LIN {X 0,Y 354.882,Z 183.277,A -85,B 0,C 180,E1 -13338.473,E2 -13338.473} C_VEL
LIN {X 0,Y 354.834,Z 183.282,A -85,B 0,C 180,E1 -13342.106,E2 -13342.106} C_VEL
LIN {X 0,Y 354.874,Z 183.277,A -85,B 0,C 180,E1 -13345.829,E2 -13345.829} C_VEL
LIN {X 0,Y 354.83,Z 183.283,A -85,B 0,C 180,E1 -13349.681,E2 -13349.681} C_VEL
LIN {X 0,Y 354.784,Z 183.288,A -85,B 0,C 180,E1 -13353.704,E2 -13353.704} C_VEL
LIN {X 0,Y 354.778,Z 183.294,A -85,B 0,C 180,E1 -13356.462,E2 -13356.462} C_VEL
LIN {X 0,Y 354.805,Z 183.286,A -85,B 0,C 180,E1 -13359.426,E2 -13359.426} C_VEL
LIN {X 0,Y 354.823,Z 183.285,A -85,B 0,C 180,E1 -13362.879,E2 -13362.879} C_VEL
LIN {X 0,Y 354.859,Z 183.284,A -85,B 0,C 180,E1 -13366.123,E2 -13366.123} C_VEL
LIN {X 0,Y 354.921,Z 183.373,A -85,B 0,C 180,E1 -13367.406,E2 -13367.406} C_VEL
LIN {X 0,Y 355.833,Z 189.151,A -85,B 0,C 180,E1 -13371.532,E2 -13371.532} C_VEL
LIN {X 0,Y 356.15,Z 192.833,A -85,B 0,C 180,E1 -13374.004,E2 -13374.004} C_VEL
LIN {X 0,Y 355.889,Z 196.663,A -85,B 0,C 180,E1 -13376.435,E2 -13376.435} C_VEL
LIN {X 0,Y 355.418,Z 202.03,A -85,B 0,C 180,E1 -13379.723,E2 -13379.723} C_VEL
LIN {X 0,Y 354.813,Z 207.607,A -85,B 0,C 180,E1 -13383.043,E2 -13383.043} C_VEL
LIN {X 0,Y 354.335,Z 213.763,A -85,B 0,C 180,E1 -13386.631,E2 -13386.631} C_VEL
LIN {X 0,Y 353.966,Z 219.424,A -85,B 0,C 180,E1 -13389.822,E2 -13389.822} C_VEL
LIN {X 0,Y 356.521,Z 232.448,A -85,B 0,C 180,E1 -13390.431,E2 -13390.431} C_VEL
LIN {X 0,Y 358.255,Z 244.108,A -85,B 0,C 180,E1 -13391.153,E2 -13391.153} C_VEL
LIN {X 0,Y 359.432,Z 255.89,A -85,B 0,C 180,E1 -13392.066,E2 -13392.066} C_VEL
LIN {X 0,Y 358.43,Z 266.908,A -85,B 0,C 180,E1 -13393.044,E2 -13393.044} C_VEL
LIN {X 0,Y 357.282,Z 277.951,A -85,B 0,C 180,E1 -13394.282,E2 -13394.282} C_VEL
LIN {X 0,Y 356.249,Z 288.12,A -85,B 0,C 180,E1 -13395.726,E2 -13395.726} C_VEL
LIN {X 0,Y 355.398,Z 296.294,A -85,B 0,C 180,E1 -13397.148,E2 -13397.148} C_VEL
LIN {X 0,Y 354.483,Z 304.31,A -85,B 0,C 180,E1 -13398.856,E2 -13398.856} C_VEL
LIN {X 0,Y 354.027,Z 309.741,A -85,B 0,C 180,E1 -13400.287,E2 -13400.287} C_VEL
LIN {X 0,Y 353.611,Z 315.06,A -85,B 0,C 180,E1 -13402.004,E2 -13402.004} C_VEL
LIN {X 0,Y 353.326,Z 319.806,A -85,B 0,C 180,E1 -13404.016,E2 -13404.016} C_VEL
LIN {X 0,Y 353.279,Z 322.276,A -85,B 0,C 180,E1 -13405.437,E2 -13405.437} C_VEL
LIN {X 0,Y 353.222,Z 323.805,A -85,B 0,C 180,E1 -13406.579,E2 -13406.579} C_VEL
LIN {X 0,Y 353.216,Z 325.559,A -85,B 0,C 180,E1 -13408.861,E2 -13408.861} C_VEL
LIN {X 0,Y 353.261,Z 325.852,A -85,B 0,C 180,E1 -13410.001,E2 -13410.001} C_VEL
LIN {X 0,Y 353.202,Z 325.754,A -85,B 0,C 180,E1 -13411.141,E2 -13411.141} C_VEL
LIN {X 0,Y 353.218,Z 324.299,A -85,B 0,C 180,E1 -13413.423,E2 -13413.423} C_VEL
LIN {X 0,Y 353.26,Z 322.979,A -85,B 0,C 180,E1 -13414.565,E2 -13414.565} C_VEL
LIN {X 0,Y 353.275,Z 320.891,A -85,B 0,C 180,E1 -13415.905,E2 -13415.905} C_VEL
LIN {X 0,Y 353.624,Z 316.373,A -85,B 0,C 180,E1 -13417.997,E2 -13417.997} C_VEL
LIN {X 0,Y 354.064,Z 311.443,A -85,B 0,C 180,E1 -13419.714,E2 -13419.714} C_VEL
LIN {X 0,Y 354.713,Z 305.246,A -85,B 0,C 180,E1 -13421.428,E2 -13421.428} C_VEL
LIN {X 0,Y 355.733,Z 297.536,A -85,B 0,C 180,E1 -13423.132,E2 -13423.132} C_VEL
LIN {X 0,Y 356.656,Z 289.652,A -85,B 0,C 180,E1 -13424.551,E2 -13424.551} C_VEL
LIN {X 0,Y 357.739,Z 280.04,A -85,B 0,C 180,E1 -13425.964,E2 -13425.964} C_VEL
LIN {X 0,Y 358.966,Z 269.382,A -85,B 0,C 180,E1 -13427.224,E2 -13427.224} C_VEL
LIN {X 0,Y 360.269,Z 257.764,A -85,B 0,C 180,E1 -13428.302,E2 -13428.302} C_VEL
LIN {X 0,Y 359.648,Z 248.942,A -85,B 0,C 180,E1 -13429.032,E2 -13429.032} C_VEL
LIN {X 0,Y 357.691,Z 236.144,A -85,B 0,C 180,E1 -13429.929,E2 -13429.929} C_VEL
LIN {X 0,Y 354.901,Z 222.926,A -85,B 0,C 180,E1 -13430.652,E2 -13430.652} C_VEL
LIN {X 0,Y 354.117,Z 219.156,A -85,B 0,C 180,E1 -13430.824,E2 -13430.824} C_VEL
LIN {X 0,Y 354.533,Z 213.305,A -85,B 0,C 180,E1 -13434.235,E2 -13434.235} C_VEL
LIN {X 0,Y 355.193,Z 206.406,A -85,B 0,C 180,E1 -13438.35,E2 -13438.35} C_VEL
LIN {X 0,Y 355.767,Z 200.689,A -85,B 0,C 180,E1 -13441.849,E2 -13441.849} C_VEL
LIN {X 0,Y 356.265,Z 195.851,A -85,B 0,C 180,E1 -13444.893,E2 -13444.893} C_VEL
LIN {X 0,Y 356.142,Z 191.408,A -85,B 0,C 180,E1 -13447.875,E2 -13447.875} C_VEL
LIN {X 0,Y 355.573,Z 187.459,A -85,B 0,C 180,E1 -13450.709,E2 -13450.709} C_VEL
LIN {X 0,Y 354.87,Z 183.284,A -85,B 0,C 180,E1 -13454.037,E2 -13454.037} C_VEL
LIN {X 0,Y 354.783,Z 183.295,A -85,B 0,C 180,E1 -13457.661,E2 -13457.661} C_VEL
LIN {X 0,Y 354.804,Z 183.286,A -85,B 0,C 180,E1 -13460.665,E2 -13460.665} C_VEL
LIN {X 0,Y 354.807,Z 183.286,A -85,B 0,C 180,E1 -13464.3,E2 -13464.3} C_VEL
LIN {X 0,Y 354.769,Z 183.293,A -85,B 0,C 180,E1 -13467.665,E2 -13467.665} C_VEL
LIN {X 0,Y 354.829,Z 183.285,A -85,B 0,C 180,E1 -13471.617,E2 -13471.617} C_VEL
LIN {X 0,Y 354.882,Z 183.276,A -85,B 0,C 180,E1 -13474.171,E2 -13474.171} C_VEL
LIN {X 0,Y 354.842,Z 183.281,A -85,B 0,C 180,E1 -13477.895,E2 -13477.895} C_VEL
LIN {X 0,Y 354.905,Z 183.273,A -85,B 0,C 180,E1 -13481.89,E2 -13481.89} C_VEL
LIN {X 0,Y 354.923,Z 183.272,A -85,B 0,C 180,E1 -13485.981,E2 -13485.981} C_VEL
LIN {X 0,Y 354.962,Z 183.266,A -85,B 0,C 180,E1 -13489.736,E2 -13489.736} C_VEL
LIN {X 0,Y 355.122,Z 183.247,A -85,B 0,C 180,E1 -13493.181,E2 -13493.181} C_VEL
LIN {X 0,Y 355.22,Z 183.235,A -85,B 0,C 180,E1 -13497.732,E2 -13497.732} C_VEL
LIN {X 0,Y 355.311,Z 183.227,A -85,B 0,C 180,E1 -13500,E2 -13500} C_VEL
LIN {X 0,Y 355.231,Z 183.237,A -85,B 0,C 180,E1 -13502.268,E2 -13502.268} C_VEL
LIN {X 0,Y 355.107,Z 183.248,A -85,B 0,C 180,E1 -13506.82,E2 -13506.82} C_VEL
LIN {X 0,Y 354.936,Z 183.272,A -85,B 0,C 180,E1 -13510.266,E2 -13510.266} C_VEL
LIN {X 0,Y 354.923,Z 183.274,A -85,B 0,C 180,E1 -13514.019,E2 -13514.019} C_VEL
LIN {X 0,Y 354.905,Z 183.275,A -85,B 0,C 180,E1 -13518.11,E2 -13518.11} C_VEL
LIN {X 0,Y 354.817,Z 183.285,A -85,B 0,C 180,E1 -13522.108,E2 -13522.108} C_VEL
LIN {X 0,Y 354.882,Z 183.278,A -85,B 0,C 180,E1 -13525.829,E2 -13525.829} C_VEL
LIN {X 0,Y 354.84,Z 183.283,A -85,B 0,C 180,E1 -13529.68,E2 -13529.68} C_VEL
LIN {X 0,Y 354.794,Z 183.288,A -85,B 0,C 180,E1 -13533.704,E2 -13533.704} C_VEL
LIN {X 0,Y 354.784,Z 183.29,A -85,B 0,C 180,E1 -13536.462,E2 -13536.462} C_VEL
LIN {X 0,Y 354.815,Z 183.286,A -85,B 0,C 180,E1 -13539.426,E2 -13539.426} C_VEL
LIN {X 0,Y 354.778,Z 183.295,A -85,B 0,C 180,E1 -13542.869,E2 -13542.869} C_VEL
LIN {X 0,Y 354.759,Z 183.293,A -85,B 0,C 180,E1 -13546.105,E2 -13546.105} C_VEL
LIN {X 0,Y 354.76,Z 183.293,A -85,B 0,C 180,E1 -13549.178,E2 -13549.178} C_VEL
LIN {X 0,Y 354.78,Z 183.295,A -85,B 0,C 180,E1 -13550.664,E2 -13550.664} C_VEL
LIN {X 0,Y 354.832,Z 186.168,A -85,B 0,C 180,E1 -13553.547,E2 -13553.547} C_VEL
LIN {X 0,Y 354.659,Z 189.195,A -85,B 0,C 180,E1 -13556.335,E2 -13556.335} C_VEL
LIN {X 0,Y 354.482,Z 192.141,A -85,B 0,C 180,E1 -13558.972,E2 -13558.972} C_VEL
LIN {X 0,Y 354.191,Z 196.682,A -85,B 0,C 180,E1 -13562.848,E2 -13562.848} C_VEL
LIN {X 0,Y 353.95,Z 201.172,A -85,B 0,C 180,E1 -13566.603,E2 -13566.603} C_VEL
LIN {X 0,Y 353.95,Z 202.182,A -85,B 0,C 180,E1 -13567.251,E2 -13567.251} C_VEL
LIN {X 0,Y 357.587,Z 215.375,A -85,B 0,C 180,E1 -13568.003,E2 -13568.003} C_VEL
LIN {X 0,Y 360.185,Z 227.262,A -85,B 0,C 180,E1 -13568.849,E2 -13568.849} C_VEL
LIN {X 0,Y 361.236,Z 233.939,A -85,B 0,C 180,E1 -13569.394,E2 -13569.394} C_VEL
LIN {X 0,Y 360.34,Z 245.219,A -85,B 0,C 180,E1 -13570.35,E2 -13570.35} C_VEL
LIN {X 0,Y 359.164,Z 255.669,A -85,B 0,C 180,E1 -13571.46,E2 -13571.46} C_VEL
LIN {X 0,Y 358.183,Z 264.323,A -85,B 0,C 180,E1 -13572.59,E2 -13572.59} C_VEL
LIN {X 0,Y 357.055,Z 273.249,A -85,B 0,C 180,E1 -13574.005,E2 -13574.005} C_VEL
LIN {X 0,Y 356.024,Z 280.897,A -85,B 0,C 180,E1 -13575.485,E2 -13575.485} C_VEL
LIN {X 0,Y 355.353,Z 287.833,A -85,B 0,C 180,E1 -13577.144,E2 -13577.144} C_VEL
LIN {X 0,Y 354.548,Z 292.713,A -85,B 0,C 180,E1 -13578.567,E2 -13578.567} C_VEL
LIN {X 0,Y 354.064,Z 297.443,A -85,B 0,C 180,E1 -13580.286,E2 -13580.286} C_VEL
LIN {X 0,Y 353.701,Z 301.063,A -85,B 0,C 180,E1 -13582.005,E2 -13582.005} C_VEL
LIN {X 0,Y 353.438,Z 303.835,A -85,B 0,C 180,E1 -13583.85,E2 -13583.85} C_VEL
LIN {X 0,Y 353.344,Z 305.343,A -85,B 0,C 180,E1 -13585.436,E2 -13585.436} C_VEL
LIN {X 0,Y 353.22,Z 306.197,A -85,B 0,C 180,E1 -13587.719,E2 -13587.719} C_VEL
LIN {X 0,Y 353.247,Z 306.014,A -85,B 0,C 180,E1 -13588.859,E2 -13588.859} C_VEL
LIN {X 0,Y 353.323,Z 304.47,A -85,B 0,C 180,E1 -13591.139,E2 -13591.139} C_VEL
LIN {X 0,Y 353.446,Z 303.118,A -85,B 0,C 180,E1 -13592.278,E2 -13592.278} C_VEL
LIN {X 0,Y 353.698,Z 300.262,A -85,B 0,C 180,E1 -13593.987,E2 -13593.987} C_VEL
LIN {X 0,Y 354.015,Z 296.392,A -85,B 0,C 180,E1 -13595.695,E2 -13595.695} C_VEL
LIN {X 0,Y 354.607,Z 290.369,A -85,B 0,C 180,E1 -13597.707,E2 -13597.707} C_VEL
LIN {X 0,Y 355.358,Z 282.686,A -85,B 0,C 180,E1 -13599.676,E2 -13599.676} C_VEL
LIN {X 0,Y 356.41,Z 274.259,A -85,B 0,C 180,E1 -13601.371,E2 -13601.371} C_VEL
LIN {X 0,Y 357.361,Z 265.595,A -85,B 0,C 180,E1 -13602.781,E2 -13602.781} C_VEL
LIN {X 0,Y 358.392,Z 254.93,A -85,B 0,C 180,E1 -13604.187,E2 -13604.187} C_VEL
LIN {X 0,Y 359.149,Z 247.136,A -85,B 0,C 180,E1 -13605.026,E2 -13605.026} C_VEL
LIN {X 0,Y 359.996,Z 236.685,A -85,B 0,C 180,E1 -13605.955,E2 -13605.955} C_VEL
LIN {X 0,Y 360.221,Z 231.766,A -85,B 0,C 180,E1 -13606.329,E2 -13606.329} C_VEL
LIN {X 0,Y 357.967,Z 218.896,A -85,B 0,C 180,E1 -13607.272,E2 -13607.272} C_VEL
LIN {X 0,Y 355.034,Z 206.448,A -85,B 0,C 180,E1 -13607.984,E2 -13607.984} C_VEL
LIN {X 0,Y 353.877,Z 201.884,A -85,B 0,C 180,E1 -13608.203,E2 -13608.203} C_VEL
LIN {X 0,Y 354.034,Z 198.323,A -85,B 0,C 180,E1 -13611.09,E2 -13611.09} C_VEL
LIN {X 0,Y 354.178,Z 194.062,A -85,B 0,C 180,E1 -13614.624,E2 -13614.624} C_VEL
LIN {X 0,Y 354.345,Z 191.093,A -85,B 0,C 180,E1 -13617.138,E2 -13617.138} C_VEL
LIN {X 0,Y 354.528,Z 188.187,A -85,B 0,C 180,E1 -13619.705,E2 -13619.705} C_VEL
LIN {X 0,Y 354.681,Z 185.272,A -85,B 0,C 180,E1 -13622.341,E2 -13622.341} C_VEL
LIN {X 0,Y 354.679,Z 183.814,A -85,B 0,C 180,E1 -13623.695,E2 -13623.695} C_VEL
LIN {X 0,Y 354.781,Z 183.293,A -85,B 0,C 180,E1 -13625.689,E2 -13625.689} C_VEL
LIN {X 0,Y 354.814,Z 183.291,A -85,B 0,C 180,E1 -13629.421,E2 -13629.421} C_VEL
LIN {X 0,Y 354.792,Z 183.291,A -85,B 0,C 180,E1 -13629.653,E2 -13629.653} C_VEL
LIN {X 0,Y 354.069,Z 183.379,A -85,B 0,C 180,E1 -13630.6,E2 -13630.6} C_VEL
LIN {X 0,Y 351.169,Z 183.739,A -85,B 0,C 180,E1 -13632.138,E2 -13632.138} C_VEL
LIN {X 0,Y 348.776,Z 184.042,A -85,B 0,C 180,E1 -13633.384,E2 -13633.384} C_VEL
LIN {X 0,Y 347.801,Z 184.159,A -85,B 0,C 180,E1 -13634.348,E2 -13634.348} C_VEL
LIN {X 0,Y 347.748,Z 184.166,A -85,B 0,C 180,E1 -13634.674,E2 -13634.674} C_VEL
LIN {X 0,Y 347.768,Z 184.163,A -85,B 0,C 180,E1 -13638.388,E2 -13638.388} C_VEL
LIN {X 0,Y 347.756,Z 184.164,A -85,B 0,C 180,E1 -13642.008,E2 -13642.008} C_VEL
LIN {X 0,Y 347.724,Z 184.169,A -85,B 0,C 180,E1 -13645.533,E2 -13645.533} C_VEL
LIN {X 0,Y 347.742,Z 184.166,A -85,B 0,C 180,E1 -13649.651,E2 -13649.651} C_VEL
LIN {X 0,Y 347.828,Z 184.16,A -85,B 0,C 180,E1 -13652.743,E2 -13652.743} C_VEL
LIN {X 0,Y 347.778,Z 184.163,A -85,B 0,C 180,E1 -13656.161,E2 -13656.161} C_VEL
LIN {X 0,Y 347.812,Z 184.156,A -85,B 0,C 180,E1 -13659.909,E2 -13659.909} C_VEL
LIN {X 0,Y 347.84,Z 184.159,A -85,B 0,C 180,E1 -13662.358,E2 -13662.358} C_VEL
LIN {X 0,Y 347.87,Z 184.153,A -85,B 0,C 180,E1 -13665.969,E2 -13665.969} C_VEL
LIN {X 0,Y 347.917,Z 184.144,A -85,B 0,C 180,E1 -13669.525,E2 -13669.525} C_VEL
LIN {X 0,Y 348.048,Z 184.132,A -85,B 0,C 180,E1 -13671.874,E2 -13671.874} C_VEL
LIN {X 0,Y 348.048,Z 184.131,A -85,B 0,C 180,E1 -13674.205,E2 -13674.205} C_VEL
LIN {X 0,Y 348.176,Z 184.115,A -85,B 0,C 180,E1 -13677.686,E2 -13677.686} C_VEL
LIN {X 0,Y 348.274,Z 184.103,A -85,B 0,C 180,E1 -13680,E2 -13680} C_VEL
LIN {X 0,Y 348.185,Z 184.111,A -85,B 0,C 180,E1 -13682.313,E2 -13682.313} C_VEL
LIN {X 0,Y 348.08,Z 184.125,A -85,B 0,C 180,E1 -13686.958,E2 -13686.958} C_VEL
LIN {X 0,Y 347.942,Z 184.145,A -85,B 0,C 180,E1 -13689.299,E2 -13689.299} C_VEL
LIN {X 0,Y 347.865,Z 184.152,A -85,B 0,C 180,E1 -13692.84,E2 -13692.84} C_VEL
LIN {X 0,Y 347.809,Z 184.157,A -85,B 0,C 180,E1 -13696.433,E2 -13696.433} C_VEL
LIN {X 0,Y 347.835,Z 184.157,A -85,B 0,C 180,E1 -13698.861,E2 -13698.861} C_VEL
LIN {X 0,Y 347.796,Z 184.16,A -85,B 0,C 180,E1 -13701.651,E2 -13701.651} C_VEL
LIN {X 0,Y 347.792,Z 184.164,A -85,B 0,C 180,E1 -13705.11,E2 -13705.11} C_VEL
LIN {X 0,Y 347.786,Z 184.16,A -85,B 0,C 180,E1 -13707.696,E2 -13707.696} C_VEL
LIN {X 0,Y 347.74,Z 184.167,A -85,B 0,C 180,E1 -13710.349,E2 -13710.349} C_VEL
LIN {X 0,Y 347.723,Z 184.172,A -85,B 0,C 180,E1 -13714.466,E2 -13714.466} C_VEL
LIN {X 0,Y 347.755,Z 184.165,A -85,B 0,C 180,E1 -13717.991,E2 -13717.991} C_VEL
LIN {X 0,Y 347.766,Z 184.163,A -85,B 0,C 180,E1 -13721.612,E2 -13721.612} C_VEL
LIN {X 0,Y 347.814,Z 184.161,A -85,B 0,C 180,E1 -13725.009,E2 -13725.009} C_VEL
LIN {X 0,Y 347.834,Z 184.193,A -85,B 0,C 180,E1 -13727.055,E2 -13727.055} C_VEL
LIN {X 0,Y 348.484,Z 188.205,A -85,B 0,C 180,E1 -13730.028,E2 -13730.028} C_VEL
LIN {X 0,Y 349.044,Z 192.193,A -85,B 0,C 180,E1 -13732.844,E2 -13732.844} C_VEL
LIN {X 0,Y 349.112,Z 195.414,A -85,B 0,C 180,E1 -13734.993,E2 -13734.993} C_VEL
LIN {X 0,Y 348.55,Z 200.76,A -85,B 0,C 180,E1 -13738.386,E2 -13738.386} C_VEL
LIN {X 0,Y 347.97,Z 206.1,A -85,B 0,C 180,E1 -13741.668,E2 -13741.668} C_VEL
LIN {X 0,Y 347.399,Z 212.577,A -85,B 0,C 180,E1 -13745.556,E2 -13745.556} C_VEL
LIN {X 0,Y 346.95,Z 219.138,A -85,B 0,C 180,E1 -13749.413,E2 -13749.413} C_VEL
LIN {X 0,Y 349.559,Z 232.284,A -85,B 0,C 180,E1 -13750.046,E2 -13750.046} C_VEL
LIN {X 0,Y 351.386,Z 244.489,A -85,B 0,C 180,E1 -13750.827,E2 -13750.827} C_VEL
LIN {X 0,Y 352.543,Z 255.477,A -85,B 0,C 180,E1 -13751.703,E2 -13751.703} C_VEL
LIN {X 0,Y 351.622,Z 266.542,A -85,B 0,C 180,E1 -13752.706,E2 -13752.706} C_VEL
LIN {X 0,Y 350.49,Z 276.804,A -85,B 0,C 180,E1 -13753.863,E2 -13753.863} C_VEL
LIN {X 0,Y 349.569,Z 286.016,A -85,B 0,C 180,E1 -13755.149,E2 -13755.149} C_VEL
LIN {X 0,Y 348.646,Z 294.515,A -85,B 0,C 180,E1 -13756.598,E2 -13756.598} C_VEL
LIN {X 0,Y 347.601,Z 302.801,A -85,B 0,C 180,E1 -13758.337,E2 -13758.337} C_VEL
LIN {X 0,Y 347.004,Z 309.484,A -85,B 0,C 180,E1 -13760.088,E2 -13760.088} C_VEL
LIN {X 0,Y 346.551,Z 314.814,A -85,B 0,C 180,E1 -13761.84,E2 -13761.84} C_VEL
LIN {X 0,Y 346.285,Z 318.965,A -85,B 0,C 180,E1 -13763.593,E2 -13763.593} C_VEL
LIN {X 0,Y 346.177,Z 322.052,A -85,B 0,C 180,E1 -13765.343,E2 -13765.343} C_VEL
LIN {X 0,Y 346.146,Z 323.588,A -85,B 0,C 180,E1 -13766.509,E2 -13766.509} C_VEL
LIN {X 0,Y 346.116,Z 325.354,A -85,B 0,C 180,E1 -13768.837,E2 -13768.837} C_VEL
LIN {X 0,Y 346.164,Z 325.652,A -85,B 0,C 180,E1 -13770.001,E2 -13770.001} C_VEL
LIN {X 0,Y 346.103,Z 325.56,A -85,B 0,C 180,E1 -13771.164,E2 -13771.164} C_VEL
LIN {X 0,Y 346.083,Z 325.039,A -85,B 0,C 180,E1 -13772.328,E2 -13772.328} C_VEL
LIN {X 0,Y 346.141,Z 324.118,A -85,B 0,C 180,E1 -13773.493,E2 -13773.493} C_VEL
LIN {X 0,Y 346.158,Z 322.801,A -85,B 0,C 180,E1 -13774.659,E2 -13774.659} C_VEL
LIN {X 0,Y 346.24,Z 320.018,A -85,B 0,C 180,E1 -13776.41,E2 -13776.41} C_VEL
LIN {X 0,Y 346.568,Z 316.216,A -85,B 0,C 180,E1 -13778.161,E2 -13778.161} C_VEL
LIN {X 0,Y 347.045,Z 311.297,A -85,B 0,C 180,E1 -13779.912,E2 -13779.912} C_VEL
LIN {X 0,Y 347.723,Z 305.112,A -85,B 0,C 180,E1 -13781.661,E2 -13781.661} C_VEL
LIN {X 0,Y 348.802,Z 297.424,A -85,B 0,C 180,E1 -13783.398,E2 -13783.398} C_VEL
LIN {X 0,Y 349.754,Z 289.558,A -85,B 0,C 180,E1 -13784.844,E2 -13784.844} C_VEL
LIN {X 0,Y 350.918,Z 279.968,A -85,B 0,C 180,E1 -13786.283,E2 -13786.283} C_VEL
LIN {X 0,Y 352.182,Z 269.336,A -85,B 0,C 180,E1 -13787.567,E2 -13787.567} C_VEL
LIN {X 0,Y 353.484,Z 257.832,A -85,B 0,C 180,E1 -13788.661,E2 -13788.661} C_VEL
LIN {X 0,Y 352.597,Z 247.927,A -85,B 0,C 180,E1 -13789.507,E2 -13789.507} C_VEL
LIN {X 0,Y 350.614,Z 235.326,A -85,B 0,C 180,E1 -13790.398,E2 -13790.398} C_VEL
LIN {X 0,Y 347.89,Z 222.697,A -85,B 0,C 180,E1 -13791.109,E2 -13791.109} C_VEL
LIN {X 0,Y 347.112,Z 218.946,A -85,B 0,C 180,E1 -13791.294,E2 -13791.294} C_VEL
LIN {X 0,Y 347.623,Z 212.519,A -85,B 0,C 180,E1 -13795.122,E2 -13795.122} C_VEL
LIN {X 0,Y 348.231,Z 206.276,A -85,B 0,C 180,E1 -13798.97,E2 -13798.97} C_VEL
LIN {X 0,Y 348.784,Z 201.152,A -85,B 0,C 180,E1 -13802.188,E2 -13802.188} C_VEL
LIN {X 0,Y 349.199,Z 197.717,A -85,B 0,C 180,E1 -13804.394,E2 -13804.394} C_VEL
LIN {X 0,Y 349.222,Z 193.647,A -85,B 0,C 180,E1 -13807.136,E2 -13807.136} C_VEL
LIN {X 0,Y 348.715,Z 189.456,A -85,B 0,C 180,E1 -13810.158,E2 -13810.158} C_VEL
LIN {X 0,Y 348.029,Z 185.279,A -85,B 0,C 180,E1 -13813.367,E2 -13813.367} C_VEL
LIN {X 0,Y 347.841,Z 184.157,A -85,B 0,C 180,E1 -13814.378,E2 -13814.378} C_VEL
LIN {X 0,Y 347.738,Z 184.168,A -85,B 0,C 180,E1 -13818.396,E2 -13818.396} C_VEL
LIN {X 0,Y 347.759,Z 184.165,A -85,B 0,C 180,E1 -13822.01,E2 -13822.01} C_VEL
LIN {X 0,Y 347.73,Z 184.172,A -85,B 0,C 180,E1 -13825.535,E2 -13825.535} C_VEL
LIN {X 0,Y 347.726,Z 184.168,A -85,B 0,C 180,E1 -13828.299,E2 -13828.299} C_VEL
LIN {X 0,Y 347.761,Z 184.168,A -85,B 0,C 180,E1 -13830.986,E2 -13830.986} C_VEL
LIN {X 0,Y 347.814,Z 184.158,A -85,B 0,C 180,E1 -13833.606,E2 -13833.606} C_VEL
LIN {X 0,Y 347.785,Z 184.161,A -85,B 0,C 180,E1 -13836.162,E2 -13836.162} C_VEL
LIN {X 0,Y 347.82,Z 184.156,A -85,B 0,C 180,E1 -13839.91,E2 -13839.91} C_VEL
LIN {X 0,Y 347.848,Z 184.155,A -85,B 0,C 180,E1 -13842.358,E2 -13842.358} C_VEL
LIN {X 0,Y 347.879,Z 184.149,A -85,B 0,C 180,E1 -13845.97,E2 -13845.97} C_VEL
LIN {X 0,Y 347.912,Z 184.144,A -85,B 0,C 180,E1 -13849.525,E2 -13849.525} C_VEL
LIN {X 0,Y 348.085,Z 184.124,A -85,B 0,C 180,E1 -13853.042,E2 -13853.042} C_VEL
LIN {X 0,Y 348.183,Z 184.112,A -85,B 0,C 180,E1 -13857.687,E2 -13857.687} C_VEL
LIN {X 0,Y 348.263,Z 184.105,A -85,B 0,C 180,E1 -13860,E2 -13860} C_VEL
LIN {X 0,Y 348.195,Z 184.113,A -85,B 0,C 180,E1 -13862.314,E2 -13862.314} C_VEL
LIN {X 0,Y 348.072,Z 184.124,A -85,B 0,C 180,E1 -13866.959,E2 -13866.959} C_VEL
LIN {X 0,Y 347.876,Z 184.15,A -85,B 0,C 180,E1 -13870.476,E2 -13870.476} C_VEL
LIN {X 0,Y 347.881,Z 184.15,A -85,B 0,C 180,E1 -13874.151,E2 -13874.151} C_VEL
LIN {X 0,Y 347.874,Z 184.15,A -85,B 0,C 180,E1 -13878.292,E2 -13878.292} C_VEL
LIN {X 0,Y 347.771,Z 184.167,A -85,B 0,C 180,E1 -13881.636,E2 -13881.636} C_VEL
LIN {X 0,Y 347.796,Z 184.162,A -85,B 0,C 180,E1 -13885.11,E2 -13885.11} C_VEL
LIN {X 0,Y 347.796,Z 184.161,A -85,B 0,C 180,E1 -13887.696,E2 -13887.696} C_VEL
LIN {X 0,Y 347.75,Z 184.165,A -85,B 0,C 180,E1 -13890.348,E2 -13890.348} C_VEL
LIN {X 0,Y 347.732,Z 184.168,A -85,B 0,C 180,E1 -13894.466,E2 -13894.466} C_VEL
LIN {X 0,Y 347.762,Z 184.163,A -85,B 0,C 180,E1 -13897.99,E2 -13897.99} C_VEL
LIN {X 0,Y 347.741,Z 184.166,A -85,B 0,C 180,E1 -13901.832,E2 -13901.832} C_VEL
LIN {X 0,Y 347.697,Z 184.175,A -85,B 0,C 180,E1 -13905.029,E2 -13905.029} C_VEL
LIN {X 0,Y 347.735,Z 184.171,A -85,B 0,C 180,E1 -13908.401,E2 -13908.401} C_VEL
LIN {X 0,Y 347.696,Z 184.175,A -85,B 0,C 180,E1 -13910.184,E2 -13910.184} C_VEL
LIN {X 0,Y 347.808,Z 185.625,A -85,B 0,C 180,E1 -13912.005,E2 -13912.005} C_VEL
LIN {X 0,Y 347.783,Z 187.796,A -85,B 0,C 180,E1 -13914.126,E2 -13914.126} C_VEL
LIN {X 0,Y 347.555,Z 190.776,A -85,B 0,C 180,E1 -13916.911,E2 -13916.911} C_VEL
LIN {X 0,Y 347.3,Z 194.765,A -85,B 0,C 180,E1 -13920.477,E2 -13920.477} C_VEL
LIN {X 0,Y 347.11,Z 198.332,A -85,B 0,C 180,E1 -13923.55,E2 -13923.55} C_VEL
LIN {X 0,Y 346.898,Z 202.133,A -85,B 0,C 180,E1 -13926.764,E2 -13926.764} C_VEL
LIN {X 0,Y 350.972,Z 217.133,A -85,B 0,C 180,E1 -13927.669,E2 -13927.669} C_VEL
LIN {X 0,Y 353.362,Z 227.998,A -85,B 0,C 180,E1 -13928.481,E2 -13928.481} C_VEL
LIN {X 0,Y 354.469,Z 235.184,A -85,B 0,C 180,E1 -13929.092,E2 -13929.092} C_VEL
LIN {X 0,Y 353.492,Z 246.676,A -85,B 0,C 180,E1 -13930.111,E2 -13930.111} C_VEL
LIN {X 0,Y 352.12,Z 258.029,A -85,B 0,C 180,E1 -13931.377,E2 -13931.377} C_VEL
LIN {X 0,Y 351.184,Z 266.316,A -85,B 0,C 180,E1 -13932.532,E2 -13932.532} C_VEL
LIN {X 0,Y 349.975,Z 274.941,A -85,B 0,C 180,E1 -13933.972,E2 -13933.972} C_VEL
LIN {X 0,Y 348.913,Z 283.031,A -85,B 0,C 180,E1 -13935.652,E2 -13935.652} C_VEL
LIN {X 0,Y 348.068,Z 290.003,A -85,B 0,C 180,E1 -13937.464,E2 -13937.464} C_VEL
LIN {X 0,Y 347.366,Z 294.556,A -85,B 0,C 180,E1 -13938.918,E2 -13938.918} C_VEL
LIN {X 0,Y 346.901,Z 298.916,A -85,B 0,C 180,E1 -13940.673,E2 -13940.673} C_VEL
LIN {X 0,Y 346.647,Z 301.219,A -85,B 0,C 180,E1 -13941.841,E2 -13941.841} C_VEL
LIN {X 0,Y 346.366,Z 304.164,A -85,B 0,C 180,E1 -13943.854,E2 -13943.854} C_VEL
LIN {X 0,Y 346.258,Z 305.525,A -85,B 0,C 180,E1 -13945.343,E2 -13945.343} C_VEL
LIN {X 0,Y 346.129,Z 306.392,A -85,B 0,C 180,E1 -13947.672,E2 -13947.672} C_VEL
LIN {X 0,Y 346.148,Z 306.222,A -85,B 0,C 180,E1 -13948.836,E2 -13948.836} C_VEL
LIN {X 0,Y 346.229,Z 304.69,A -85,B 0,C 180,E1 -13951.162,E2 -13951.162} C_VEL
LIN {X 0,Y 346.354,Z 303.344,A -85,B 0,C 180,E1 -13952.325,E2 -13952.325} C_VEL
LIN {X 0,Y 346.615,Z 300.502,A -85,B 0,C 180,E1 -13954.068,E2 -13954.068} C_VEL
LIN {X 0,Y 346.979,Z 296.645,A -85,B 0,C 180,E1 -13955.811,E2 -13955.811} C_VEL
LIN {X 0,Y 347.534,Z 291.103,A -85,B 0,C 180,E1 -13957.731,E2 -13957.731} C_VEL
LIN {X 0,Y 348.244,Z 284.203,A -85,B 0,C 180,E1 -13959.583,E2 -13959.583} C_VEL
LIN {X 0,Y 349.265,Z 276.103,A -85,B 0,C 180,E1 -13961.313,E2 -13961.313} C_VEL
LIN {X 0,Y 350.278,Z 267.822,A -85,B 0,C 180,E1 -13962.749,E2 -13962.749} C_VEL
LIN {X 0,Y 351.333,Z 257.645,A -85,B 0,C 180,E1 -13964.183,E2 -13964.183} C_VEL
LIN {X 0,Y 352.326,Z 247.557,A -85,B 0,C 180,E1 -13965.324,E2 -13965.324} C_VEL
LIN {X 0,Y 353.184,Z 237.263,A -85,B 0,C 180,E1 -13966.263,E2 -13966.263} C_VEL
LIN {X 0,Y 353.364,Z 232.64,A -85,B 0,C 180,E1 -13966.628,E2 -13966.628} C_VEL
LIN {X 0,Y 351.104,Z 219.541,A -85,B 0,C 180,E1 -13967.619,E2 -13967.619} C_VEL
LIN {X 0,Y 348.063,Z 206.909,A -85,B 0,C 180,E1 -13968.373,E2 -13968.373} C_VEL
LIN {X 0,Y 346.817,Z 202.068,A -85,B 0,C 180,E1 -13968.615,E2 -13968.615} C_VEL
LIN {X 0,Y 346.979,Z 198.735,A -85,B 0,C 180,E1 -13971.38,E2 -13971.38} C_VEL
LIN {X 0,Y 347.162,Z 194.278,A -85,B 0,C 180,E1 -13975.156,E2 -13975.156} C_VEL
LIN {X 0,Y 347.326,Z 191.291,A -85,B 0,C 180,E1 -13977.733,E2 -13977.733} C_VEL
LIN {X 0,Y 347.52,Z 188.364,A -85,B 0,C 180,E1 -13980.367,E2 -13980.367} C_VEL
LIN {X 0,Y 347.625,Z 185.462,A -85,B 0,C 180,E1 -13983.08,E2 -13983.08} C_VEL
LIN {X 0,Y 347.642,Z 184.182,A -85,B 0,C 180,E1 -13984.472,E2 -13984.472} C_VEL
LIN {X 0,Y 347.745,Z 184.17,A -85,B 0,C 180,E1 -13987.319,E2 -13987.319} C_VEL
LIN {X 0,Y 347.72,Z 184.168,A -85,B 0,C 180,E1 -13990.294,E2 -13990.294} C_VEL
LIN {X 0,Y 347.716,Z 184.174,A -85,B 0,C 180,E1 -13993.404,E2 -13993.404} C_VEL
LIN {X 0,Y 347.748,Z 184.166,A -85,B 0,C 180,E1 -13994.674,E2 -13994.674} C_VEL
LIN {X 0,Y 347.161,Z 184.244,A -85,B 0,C 180,E1 -13995.641,E2 -13995.641} C_VEL
LIN {X 0,Y 344.366,Z 184.594,A -85,B 0,C 180,E1 -13997.215,E2 -13997.215} C_VEL
LIN {X 0,Y 341.93,Z 184.895,A -85,B 0,C 180,E1 -13998.489,E2 -13998.489} C_VEL
LIN {X 0,Y 340.847,Z 185.028,A -85,B 0,C 180,E1 -13999.475,E2 -13999.475} C_VEL
LIN {X 0,Y 340.741,Z 185.038,A -85,B 0,C 180,E1 -13999.809,E2 -13999.809} C_VEL
LIN {X 0,Y 340.691,Z 185.045,A -85,B 0,C 180,E1 -14003.557,E2 -14003.557} C_VEL
LIN {X 0,Y 340.672,Z 185.047,A -85,B 0,C 180,E1 -14006.151,E2 -14006.151} C_VEL
LIN {X 0,Y 340.753,Z 185.038,A -85,B 0,C 180,E1 -14010.33,E2 -14010.33} C_VEL
LIN {X 0,Y 340.781,Z 185.035,A -85,B 0,C 180,E1 -14013.018,E2 -14013.018} C_VEL
LIN {X 0,Y 340.719,Z 185.04,A -85,B 0,C 180,E1 -14016.926,E2 -14016.926} C_VEL
LIN {X 0,Y 340.778,Z 185.034,A -85,B 0,C 180,E1 -14020.732,E2 -14020.732} C_VEL
LIN {X 0,Y 340.761,Z 185.035,A -85,B 0,C 180,E1 -14023.217,E2 -14023.217} C_VEL
LIN {X 0,Y 340.822,Z 185.028,A -85,B 0,C 180,E1 -14026.889,E2 -14026.889} C_VEL
LIN {X 0,Y 340.938,Z 185.015,A -85,B 0,C 180,E1 -14030.508,E2 -14030.508} C_VEL
LIN {X 0,Y 341.057,Z 184.998,A -85,B 0,C 180,E1 -14032.898,E2 -14032.898} C_VEL
LIN {X 0,Y 341.139,Z 184.991,A -85,B 0,C 180,E1 -14037.638,E2 -14037.638} C_VEL
LIN {X 0,Y 341.225,Z 184.981,A -85,B 0,C 180,E1 -14040,E2 -14040} C_VEL
LIN {X 0,Y 341.148,Z 184.988,A -85,B 0,C 180,E1 -14042.361,E2 -14042.361} C_VEL
LIN {X 0,Y 341.049,Z 185.001,A -85,B 0,C 180,E1 -14047.102,E2 -14047.102} C_VEL
LIN {X 0,Y 340.849,Z 185.025,A -85,B 0,C 180,E1 -14050.694,E2 -14050.694} C_VEL
LIN {X 0,Y 340.836,Z 185.026,A -85,B 0,C 180,E1 -14054.326,E2 -14054.326} C_VEL
LIN {X 0,Y 340.811,Z 185.03,A -85,B 0,C 180,E1 -14058.468,E2 -14058.468} C_VEL
LIN {X 0,Y 340.737,Z 185.039,A -85,B 0,C 180,E1 -14061.862,E2 -14061.862} C_VEL
LIN {X 0,Y 340.75,Z 185.037,A -85,B 0,C 180,E1 -14065.666,E2 -14065.666} C_VEL
LIN {X 0,Y 340.717,Z 185.042,A -85,B 0,C 180,E1 -14068.322,E2 -14068.322} C_VEL
LIN {X 0,Y 340.68,Z 185.048,A -85,B 0,C 180,E1 -14071.046,E2 -14071.046} C_VEL
LIN {X 0,Y 340.697,Z 185.044,A -85,B 0,C 180,E1 -14075.281,E2 -14075.281} C_VEL
LIN {X 0,Y 340.693,Z 185.048,A -85,B 0,C 180,E1 -14078.389,E2 -14078.389} C_VEL
LIN {X 0,Y 340.707,Z 185.042,A -85,B 0,C 180,E1 -14081.306,E2 -14081.306} C_VEL
LIN {X 0,Y 340.765,Z 185.04,A -85,B 0,C 180,E1 -14084.525,E2 -14084.525} C_VEL
LIN {X 0,Y 340.8,Z 185.118,A -85,B 0,C 180,E1 -14086.781,E2 -14086.781} C_VEL
LIN {X 0,Y 341.561,Z 189.857,A -85,B 0,C 180,E1 -14090.372,E2 -14090.372} C_VEL
LIN {X 0,Y 342.072,Z 193.89,A -85,B 0,C 180,E1 -14093.252,E2 -14093.252} C_VEL
LIN {X 0,Y 342.024,Z 196.891,A -85,B 0,C 180,E1 -14095.278,E2 -14095.278} C_VEL
LIN {X 0,Y 341.443,Z 202.709,A -85,B 0,C 180,E1 -14099.034,E2 -14099.034} C_VEL
LIN {X 0,Y 340.689,Z 209.088,A -85,B 0,C 180,E1 -14103.013,E2 -14103.013} C_VEL
LIN {X 0,Y 340.159,Z 215.425,A -85,B 0,C 180,E1 -14106.889,E2 -14106.889} C_VEL
LIN {X 0,Y 339.905,Z 218.886,A -85,B 0,C 180,E1 -14108.982,E2 -14108.982} C_VEL
LIN {X 0,Y 342.626,Z 232.502,A -85,B 0,C 180,E1 -14109.665,E2 -14109.665} C_VEL
LIN {X 0,Y 344.506,Z 245.07,A -85,B 0,C 180,E1 -14110.501,E2 -14110.501} C_VEL
LIN {X 0,Y 345.691,Z 256.845,A -85,B 0,C 180,E1 -14111.481,E2 -14111.481} C_VEL
LIN {X 0,Y 344.688,Z 267.606,A -85,B 0,C 180,E1 -14112.5,E2 -14112.5} C_VEL
LIN {X 0,Y 343.41,Z 278.578,A -85,B 0,C 180,E1 -14113.812,E2 -14113.812} C_VEL
LIN {X 0,Y 342.46,Z 287.523,A -85,B 0,C 180,E1 -14115.139,E2 -14115.139} C_VEL
LIN {X 0,Y 341.327,Z 297.215,A -85,B 0,C 180,E1 -14116.911,E2 -14116.911} C_VEL
LIN {X 0,Y 340.36,Z 304.936,A -85,B 0,C 180,E1 -14118.689,E2 -14118.689} C_VEL
LIN {X 0,Y 339.79,Z 311.142,A -85,B 0,C 180,E1 -14120.477,E2 -14120.477} C_VEL
LIN {X 0,Y 339.394,Z 316.071,A -85,B 0,C 180,E1 -14122.266,E2 -14122.266} C_VEL
LIN {X 0,Y 339.134,Z 319.97,A -85,B 0,C 180,E1 -14124.111,E2 -14124.111} C_VEL
LIN {X 0,Y 339.07,Z 323.371,A -85,B 0,C 180,E1 -14126.436,E2 -14126.436} C_VEL
LIN {X 0,Y 338.999,Z 324.46,A -85,B 0,C 180,E1 -14127.625,E2 -14127.625} C_VEL
LIN {X 0,Y 339.018,Z 325.149,A -85,B 0,C 180,E1 -14128.813,E2 -14128.813} C_VEL
LIN {X 0,Y 339.066,Z 325.452,A -85,B 0,C 180,E1 -14130.001,E2 -14130.001} C_VEL
LIN {X 0,Y 339.006,Z 325.365,A -85,B 0,C 180,E1 -14131.189,E2 -14131.189} C_VEL
LIN {X 0,Y 338.997,Z 324.853,A -85,B 0,C 180,E1 -14132.377,E2 -14132.377} C_VEL
LIN {X 0,Y 339.065,Z 323.937,A -85,B 0,C 180,E1 -14133.566,E2 -14133.566} C_VEL
LIN {X 0,Y 339.111,Z 321.057,A -85,B 0,C 180,E1 -14135.85,E2 -14135.85} C_VEL
LIN {X 0,Y 339.4,Z 317.463,A -85,B 0,C 180,E1 -14137.736,E2 -14137.736} C_VEL
LIN {X 0,Y 339.827,Z 312.942,A -85,B 0,C 180,E1 -14139.523,E2 -14139.523} C_VEL
LIN {X 0,Y 340.607,Z 306.099,A -85,B 0,C 180,E1 -14141.606,E2 -14141.606} C_VEL
LIN {X 0,Y 341.677,Z 298.683,A -85,B 0,C 180,E1 -14143.379,E2 -14143.379} C_VEL
LIN {X 0,Y 342.662,Z 291.131,A -85,B 0,C 180,E1 -14144.855,E2 -14144.855} C_VEL
LIN {X 0,Y 343.905,Z 281.298,A -85,B 0,C 180,E1 -14146.424,E2 -14146.424} C_VEL
LIN {X 0,Y 345.275,Z 270.582,A -85,B 0,C 180,E1 -14147.777,E2 -14147.777} C_VEL
LIN {X 0,Y 346.654,Z 259.06,A -85,B 0,C 180,E1 -14148.928,E2 -14148.928} C_VEL
LIN {X 0,Y 345.789,Z 248.568,A -85,B 0,C 180,E1 -14149.861,E2 -14149.861} C_VEL
LIN {X 0,Y 344.062,Z 237.202,A -85,B 0,C 180,E1 -14150.714,E2 -14150.714} C_VEL
LIN {X 0,Y 341.444,Z 224.671,A -85,B 0,C 180,E1 -14151.47,E2 -14151.47} C_VEL
LIN {X 0,Y 340.093,Z 218.76,A -85,B 0,C 180,E1 -14151.76,E2 -14151.76} C_VEL
LIN {X 0,Y 340.639,Z 212.393,A -85,B 0,C 180,E1 -14155.674,E2 -14155.674} C_VEL
LIN {X 0,Y 341.326,Z 206.13,A -85,B 0,C 180,E1 -14159.613,E2 -14159.613} C_VEL
LIN {X 0,Y 342.067,Z 199.843,A -85,B 0,C 180,E1 -14163.691,E2 -14163.691} C_VEL
LIN {X 0,Y 342.233,Z 195.636,A -85,B 0,C 180,E1 -14166.549,E2 -14166.549} C_VEL
LIN {X 0,Y 341.816,Z 191.438,A -85,B 0,C 180,E1 -14169.595,E2 -14169.595} C_VEL
LIN {X 0,Y 341.157,Z 187.279,A -85,B 0,C 180,E1 -14172.826,E2 -14172.826} C_VEL
LIN {X 0,Y 340.765,Z 185.039,A -85,B 0,C 180,E1 -14174.752,E2 -14174.752} C_VEL
LIN {X 0,Y 340.674,Z 185.048,A -85,B 0,C 180,E1 -14178.689,E2 -14178.689} C_VEL
LIN {X 0,Y 340.719,Z 185.044,A -85,B 0,C 180,E1 -14181.771,E2 -14181.771} C_VEL
LIN {X 0,Y 340.709,Z 185.046,A -85,B 0,C 180,E1 -14185.594,E2 -14185.594} C_VEL
LIN {X 0,Y 340.678,Z 185.05,A -85,B 0,C 180,E1 -14188.953,E2 -14188.953} C_VEL
LIN {X 0,Y 340.775,Z 185.039,A -85,B 0,C 180,E1 -14193.018,E2 -14193.018} C_VEL
LIN {X 0,Y 340.764,Z 185.036,A -85,B 0,C 180,E1 -14195.639,E2 -14195.639} C_VEL
LIN {X 0,Y 340.764,Z 185.036,A -85,B 0,C 180,E1 -14199.475,E2 -14199.475} C_VEL
LIN {X 0,Y 340.84,Z 185.026,A -85,B 0,C 180,E1 -14201.983,E2 -14201.983} C_VEL
LIN {X 0,Y 340.834,Z 185.026,A -85,B 0,C 180,E1 -14205.716,E2 -14205.716} C_VEL
LIN {X 0,Y 340.855,Z 185.024,A -85,B 0,C 180,E1 -14209.306,E2 -14209.306} C_VEL
LIN {X 0,Y 341.051,Z 185.001,A -85,B 0,C 180,E1 -14212.898,E2 -14212.898} C_VEL
LIN {X 0,Y 341.145,Z 184.988,A -85,B 0,C 180,E1 -14217.639,E2 -14217.639} C_VEL
LIN {X 0,Y 341.215,Z 184.983,A -85,B 0,C 180,E1 -14220,E2 -14220} C_VEL
LIN {X 0,Y 341.157,Z 184.989,A -85,B 0,C 180,E1 -14222.362,E2 -14222.362} C_VEL
LIN {X 0,Y 341.04,Z 185.001,A -85,B 0,C 180,E1 -14227.103,E2 -14227.103} C_VEL
LIN {X 0,Y 340.827,Z 185.027,A -85,B 0,C 180,E1 -14230.696,E2 -14230.696} C_VEL
LIN {X 0,Y 340.846,Z 185.025,A -85,B 0,C 180,E1 -14234.326,E2 -14234.326} C_VEL
LIN {X 0,Y 340.821,Z 185.028,A -85,B 0,C 180,E1 -14238.468,E2 -14238.468} C_VEL
LIN {X 0,Y 340.738,Z 185.041,A -85,B 0,C 180,E1 -14241.858,E2 -14241.858} C_VEL
LIN {X 0,Y 340.757,Z 185.039,A -85,B 0,C 180,E1 -14245.666,E2 -14245.666} C_VEL
LIN {X 0,Y 340.727,Z 185.04,A -85,B 0,C 180,E1 -14248.321,E2 -14248.321} C_VEL
LIN {X 0,Y 340.69,Z 185.048,A -85,B 0,C 180,E1 -14251.046,E2 -14251.046} C_VEL
LIN {X 0,Y 340.706,Z 185.046,A -85,B 0,C 180,E1 -14255.281,E2 -14255.281} C_VEL
LIN {X 0,Y 340.698,Z 185.044,A -85,B 0,C 180,E1 -14258.387,E2 -14258.387} C_VEL
LIN {X 0,Y 340.689,Z 185.044,A -85,B 0,C 180,E1 -14262.047,E2 -14262.047} C_VEL
LIN {X 0,Y 340.644,Z 185.052,A -85,B 0,C 180,E1 -14266.229,E2 -14266.229} C_VEL
LIN {X 0,Y 340.665,Z 185.053,A -85,B 0,C 180,E1 -14268.69,E2 -14268.69} C_VEL
LIN {X 0,Y 340.646,Z 185.054,A -85,B 0,C 180,E1 -14270.242,E2 -14270.242} C_VEL
LIN {X 0,Y 340.768,Z 187.941,A -85,B 0,C 180,E1 -14273.268,E2 -14273.268} C_VEL
LIN {X 0,Y 340.583,Z 190.914,A -85,B 0,C 180,E1 -14276.143,E2 -14276.143} C_VEL
LIN {X 0,Y 340.351,Z 193.942,A -85,B 0,C 180,E1 -14278.922,E2 -14278.922} C_VEL
LIN {X 0,Y 340.093,Z 198.165,A -85,B 0,C 180,E1 -14282.698,E2 -14282.698} C_VEL
LIN {X 0,Y 339.89,Z 202.465,A -85,B 0,C 180,E1 -14286.304,E2 -14286.304} C_VEL
LIN {X 0,Y 343.578,Z 215.689,A -85,B 0,C 180,E1 -14287.103,E2 -14287.103} C_VEL
LIN {X 0,Y 346.309,Z 227.532,A -85,B 0,C 180,E1 -14288,E2 -14288} C_VEL
LIN {X 0,Y 347.725,Z 236.381,A -85,B 0,C 180,E1 -14288.779,E2 -14288.779} C_VEL
LIN {X 0,Y 346.642,Z 247.925,A -85,B 0,C 180,E1 -14289.839,E2 -14289.839} C_VEL
LIN {X 0,Y 345.232,Z 259.182,A -85,B 0,C 180,E1 -14291.146,E2 -14291.146} C_VEL
LIN {X 0,Y 344.141,Z 268.233,A -85,B 0,C 180,E1 -14292.469,E2 -14292.469} C_VEL
LIN {X 0,Y 342.927,Z 276.521,A -85,B 0,C 180,E1 -14293.939,E2 -14293.939} C_VEL
LIN {X 0,Y 341.817,Z 284.621,A -85,B 0,C 180,E1 -14295.716,E2 -14295.716} C_VEL
LIN {X 0,Y 340.932,Z 291.126,A -85,B 0,C 180,E1 -14297.5,E2 -14297.5} C_VEL
LIN {X 0,Y 340.193,Z 296.294,A -85,B 0,C 180,E1 -14299.285,E2 -14299.285} C_VEL
LIN {X 0,Y 339.734,Z 300.299,A -85,B 0,C 180,E1 -14301.074,E2 -14301.074} C_VEL
LIN {X 0,Y 339.388,Z 303.258,A -85,B 0,C 180,E1 -14302.862,E2 -14302.862} C_VEL
LIN {X 0,Y 339.219,Z 304.696,A -85,B 0,C 180,E1 -14304.054,E2 -14304.054} C_VEL
LIN {X 0,Y 339.176,Z 305.707,A -85,B 0,C 180,E1 -14305.245,E2 -14305.245} C_VEL
LIN {X 0,Y 339.105,Z 306.336,A -85,B 0,C 180,E1 -14306.435,E2 -14306.435} C_VEL
LIN {X 0,Y 339.041,Z 306.587,A -85,B 0,C 180,E1 -14307.623,E2 -14307.623} C_VEL
LIN {X 0,Y 339.049,Z 306.429,A -85,B 0,C 180,E1 -14308.812,E2 -14308.812} C_VEL
LIN {X 0,Y 339.135,Z 304.909,A -85,B 0,C 180,E1 -14311.187,E2 -14311.187} C_VEL
LIN {X 0,Y 339.263,Z 303.571,A -85,B 0,C 180,E1 -14312.374,E2 -14312.374} C_VEL
LIN {X 0,Y 339.538,Z 300.741,A -85,B 0,C 180,E1 -14314.153,E2 -14314.153} C_VEL
LIN {X 0,Y 339.944,Z 296.898,A -85,B 0,C 180,E1 -14315.932,E2 -14315.932} C_VEL
LIN {X 0,Y 340.481,Z 291.726,A -85,B 0,C 180,E1 -14317.779,E2 -14317.779} C_VEL
LIN {X 0,Y 341.253,Z 284.498,A -85,B 0,C 180,E1 -14319.781,E2 -14319.781} C_VEL
LIN {X 0,Y 342.334,Z 276.417,A -85,B 0,C 180,E1 -14321.545,E2 -14321.545} C_VEL
LIN {X 0,Y 343.378,Z 268.159,A -85,B 0,C 180,E1 -14323.009,E2 -14323.009} C_VEL
LIN {X 0,Y 344.477,Z 258.026,A -85,B 0,C 180,E1 -14324.471,E2 -14324.471} C_VEL
LIN {X 0,Y 345.515,Z 247.978,A -85,B 0,C 180,E1 -14325.633,E2 -14325.633} C_VEL
LIN {X 0,Y 346.456,Z 236.879,A -85,B 0,C 180,E1 -14326.662,E2 -14326.662} C_VEL
LIN {X 0,Y 346.533,Z 233.615,A -85,B 0,C 180,E1 -14326.93,E2 -14326.93} C_VEL
LIN {X 0,Y 344.301,Z 220.57,A -85,B 0,C 180,E1 -14327.954,E2 -14327.954} C_VEL
LIN {X 0,Y 341.244,Z 208.035,A -85,B 0,C 180,E1 -14328.746,E2 -14328.746} C_VEL
LIN {X 0,Y 339.744,Z 202.248,A -85,B 0,C 180,E1 -14329.063,E2 -14329.063} C_VEL
LIN {X 0,Y 339.917,Z 198.945,A -85,B 0,C 180,E1 -14331.846,E2 -14331.846} C_VEL
LIN {X 0,Y 340.151,Z 194.472,A -85,B 0,C 180,E1 -14335.712,E2 -14335.712} C_VEL
LIN {X 0,Y 340.328,Z 191.49,A -85,B 0,C 180,E1 -14338.354,E2 -14338.354} C_VEL
LIN {X 0,Y 340.522,Z 188.566,A -85,B 0,C 180,E1 -14341.059,E2 -14341.059} C_VEL
LIN {X 0,Y 340.59,Z 185.107,A -85,B 0,C 180,E1 -14344.371,E2 -14344.371} C_VEL
LIN {X 0,Y 340.684,Z 185.046,A -85,B 0,C 180,E1 -14346.74,E2 -14346.74} C_VEL
LIN {X 0,Y 340.676,Z 185.046,A -85,B 0,C 180,E1 -14350.244,E2 -14350.244} C_VEL
LIN {X 0,Y 340.663,Z 185.049,A -85,B 0,C 180,E1 -14353.774,E2 -14353.774} C_VEL
LIN {X 0,Y 340.723,Z 185.045,A -85,B 0,C 180,E1 -14357.102,E2 -14357.102} C_VEL
LIN {X 0,Y 340.741,Z 185.038,A -85,B 0,C 180,E1 -14359.809,E2 -14359.809} C_VEL
LIN {X 0,Y 340.017,Z 185.132,A -85,B 0,C 180,E1 -14360.795,E2 -14360.795} C_VEL
LIN {X 0,Y 337.115,Z 185.49,A -85,B 0,C 180,E1 -14362.4,E2 -14362.4} C_VEL
LIN {X 0,Y 334.712,Z 185.789,A -85,B 0,C 180,E1 -14363.7,E2 -14363.7} C_VEL
LIN {X 0,Y 333.717,Z 185.917,A -85,B 0,C 180,E1 -14364.706,E2 -14364.706} C_VEL
LIN {X 0,Y 333.654,Z 185.922,A -85,B 0,C 180,E1 -14365.047,E2 -14365.047} C_VEL
LIN {X 0,Y 333.612,Z 185.927,A -85,B 0,C 180,E1 -14368.219,E2 -14368.219} C_VEL
LIN {X 0,Y 333.689,Z 185.919,A -85,B 0,C 180,E1 -14371.025,E2 -14371.025} C_VEL
LIN {X 0,Y 333.713,Z 185.913,A -85,B 0,C 180,E1 -14373.751,E2 -14373.751} C_VEL
LIN {X 0,Y 333.701,Z 185.912,A -85,B 0,C 180,E1 -14377.91,E2 -14377.91} C_VEL
LIN {X 0,Y 333.769,Z 185.904,A -85,B 0,C 180,E1 -14381.588,E2 -14381.588} C_VEL
LIN {X 0,Y 333.782,Z 185.905,A -85,B 0,C 180,E1 -14385.575,E2 -14385.575} C_VEL
LIN {X 0,Y 333.818,Z 185.898,A -85,B 0,C 180,E1 -14389.077,E2 -14389.077} C_VEL
LIN {X 0,Y 333.999,Z 185.879,A -85,B 0,C 180,E1 -14391.53,E2 -14391.53} C_VEL
LIN {X 0,Y 334.001,Z 185.883,A -85,B 0,C 180,E1 -14393.96,E2 -14393.96} C_VEL
LIN {X 0,Y 334.076,Z 185.87,A -85,B 0,C 180,E1 -14397.588,E2 -14397.588} C_VEL
LIN {X 0,Y 334.178,Z 185.859,A -85,B 0,C 180,E1 -14400,E2 -14400} C_VEL
LIN {X 0,Y 334.11,Z 185.864,A -85,B 0,C 180,E1 -14402.411,E2 -14402.411} C_VEL
LIN {X 0,Y 333.998,Z 185.881,A -85,B 0,C 180,E1 -14407.253,E2 -14407.253} C_VEL
LIN {X 0,Y 333.811,Z 185.903,A -85,B 0,C 180,E1 -14410.922,E2 -14410.922} C_VEL
LIN {X 0,Y 333.781,Z 185.906,A -85,B 0,C 180,E1 -14414.635,E2 -14414.635} C_VEL
LIN {X 0,Y 333.771,Z 185.908,A -85,B 0,C 180,E1 -14418.657,E2 -14418.657} C_VEL
LIN {X 0,Y 333.695,Z 185.916,A -85,B 0,C 180,E1 -14422.278,E2 -14422.278} C_VEL
LIN {X 0,Y 333.712,Z 185.914,A -85,B 0,C 180,E1 -14426.248,E2 -14426.248} C_VEL
LIN {X 0,Y 333.687,Z 185.919,A -85,B 0,C 180,E1 -14428.974,E2 -14428.974} C_VEL
LIN {X 0,Y 333.621,Z 185.929,A -85,B 0,C 180,E1 -14432.589,E2 -14432.589} C_VEL
LIN {X 0,Y 333.656,Z 185.922,A -85,B 0,C 180,E1 -14436.141,E2 -14436.141} C_VEL
LIN {X 0,Y 333.663,Z 185.92,A -85,B 0,C 180,E1 -14439.19,E2 -14439.19} C_VEL
LIN {X 0,Y 333.686,Z 185.922,A -85,B 0,C 180,E1 -14442.516,E2 -14442.516} C_VEL
LIN {X 0,Y 333.776,Z 186,A -85,B 0,C 180,E1 -14446.469,E2 -14446.469} C_VEL
LIN {X 0,Y 334.517,Z 190.738,A -85,B 0,C 180,E1 -14450.154,E2 -14450.154} C_VEL
LIN {X 0,Y 334.998,Z 194.439,A -85,B 0,C 180,E1 -14452.864,E2 -14452.864} C_VEL
LIN {X 0,Y 335.045,Z 197.344,A -85,B 0,C 180,E1 -14454.893,E2 -14454.893} C_VEL
LIN {X 0,Y 334.468,Z 202.507,A -85,B 0,C 180,E1 -14458.314,E2 -14458.314} C_VEL
LIN {X 0,Y 333.785,Z 208.501,A -85,B 0,C 180,E1 -14462.169,E2 -14462.169} C_VEL
LIN {X 0,Y 333.143,Z 215.207,A -85,B 0,C 180,E1 -14466.373,E2 -14466.373} C_VEL
LIN {X 0,Y 332.905,Z 218.697,A -85,B 0,C 180,E1 -14468.542,E2 -14468.542} C_VEL
LIN {X 0,Y 335.622,Z 232.133,A -85,B 0,C 180,E1 -14469.233,E2 -14469.233} C_VEL
LIN {X 0,Y 337.511,Z 244.545,A -85,B 0,C 180,E1 -14470.077,E2 -14470.077} C_VEL
LIN {X 0,Y 338.721,Z 256.422,A -85,B 0,C 180,E1 -14471.085,E2 -14471.085} C_VEL
LIN {X 0,Y 338.372,Z 262.932,A -85,B 0,C 180,E1 -14471.693,E2 -14471.693} C_VEL
LIN {X 0,Y 337.119,Z 273.652,A -85,B 0,C 180,E1 -14472.877,E2 -14472.877} C_VEL
LIN {X 0,Y 335.967,Z 283.43,A -85,B 0,C 180,E1 -14474.222,E2 -14474.222} C_VEL
LIN {X 0,Y 334.916,Z 292.335,A -85,B 0,C 180,E1 -14475.727,E2 -14475.727} C_VEL
LIN {X 0,Y 333.84,Z 301.02,A -85,B 0,C 180,E1 -14477.54,E2 -14477.54} C_VEL
LIN {X 0,Y 333.062,Z 307.953,A -85,B 0,C 180,E1 -14479.362,E2 -14479.362} C_VEL
LIN {X 0,Y 332.452,Z 314.322,A -85,B 0,C 180,E1 -14481.492,E2 -14481.492} C_VEL
LIN {X 0,Y 332.159,Z 318.494,A -85,B 0,C 180,E1 -14483.319,E2 -14483.319} C_VEL
LIN {X 0,Y 331.986,Z 321.603,A -85,B 0,C 180,E1 -14485.144,E2 -14485.144} C_VEL
LIN {X 0,Y 331.996,Z 323.154,A -85,B 0,C 180,E1 -14486.36,E2 -14486.36} C_VEL
LIN {X 0,Y 331.916,Z 324.251,A -85,B 0,C 180,E1 -14487.574,E2 -14487.574} C_VEL
LIN {X 0,Y 331.923,Z 324.944,A -85,B 0,C 180,E1 -14488.788,E2 -14488.788} C_VEL
LIN {X 0,Y 331.969,Z 325.252,A -85,B 0,C 180,E1 -14490.001,E2 -14490.001} C_VEL
LIN {X 0,Y 331.912,Z 325.17,A -85,B 0,C 180,E1 -14491.214,E2 -14491.214} C_VEL
LIN {X 0,Y 331.915,Z 324.667,A -85,B 0,C 180,E1 -14492.428,E2 -14492.428} C_VEL
LIN {X 0,Y 331.968,Z 323.755,A -85,B 0,C 180,E1 -14493.642,E2 -14493.642} C_VEL
LIN {X 0,Y 332.005,Z 321.172,A -85,B 0,C 180,E1 -14495.782,E2 -14495.782} C_VEL
LIN {X 0,Y 332.358,Z 317.301,A -85,B 0,C 180,E1 -14497.9,E2 -14497.9} C_VEL
LIN {X 0,Y 332.803,Z 312.791,A -85,B 0,C 180,E1 -14499.726,E2 -14499.726} C_VEL
LIN {X 0,Y 333.621,Z 305.967,A -85,B 0,C 180,E1 -14501.852,E2 -14501.852} C_VEL
LIN {X 0,Y 334.752,Z 298.565,A -85,B 0,C 180,E1 -14503.662,E2 -14503.662} C_VEL
LIN {X 0,Y 335.999,Z 289.372,A -85,B 0,C 180,E1 -14505.467,E2 -14505.467} C_VEL
LIN {X 0,Y 337.268,Z 279.825,A -85,B 0,C 180,E1 -14506.961,E2 -14506.961} C_VEL
LIN {X 0,Y 338.659,Z 269.246,A -85,B 0,C 180,E1 -14508.293,E2 -14508.293} C_VEL
LIN {X 0,Y 339.886,Z 259.051,A -85,B 0,C 180,E1 -14509.319,E2 -14509.319} C_VEL
LIN {X 0,Y 338.706,Z 246.983,A -85,B 0,C 180,E1 -14510.42,E2 -14510.42} C_VEL
LIN {X 0,Y 336.602,Z 233.99,A -85,B 0,C 180,E1 -14511.377,E2 -14511.377} C_VEL
LIN {X 0,Y 333.525,Z 220.822,A -85,B 0,C 180,E1 -14512.159,E2 -14512.159} C_VEL
LIN {X 0,Y 333.093,Z 218.556,A -85,B 0,C 180,E1 -14512.278,E2 -14512.278} C_VEL
LIN {X 0,Y 333.656,Z 212.23,A -85,B 0,C 180,E1 -14516.252,E2 -14516.252} C_VEL
LIN {X 0,Y 334.435,Z 205.672,A -85,B 0,C 180,E1 -14520.504,E2 -14520.504} C_VEL
LIN {X 0,Y 335.117,Z 199.722,A -85,B 0,C 180,E1 -14524.486,E2 -14524.486} C_VEL
LIN {X 0,Y 335.27,Z 197.611,A -85,B 0,C 180,E1 -14525.938,E2 -14525.938} C_VEL
LIN {X 0,Y 334.927,Z 193.332,A -85,B 0,C 180,E1 -14529.068,E2 -14529.068} C_VEL
LIN {X 0,Y 334.217,Z 188.857,A -85,B 0,C 180,E1 -14532.609,E2 -14532.609} C_VEL
LIN {X 0,Y 333.702,Z 185.921,A -85,B 0,C 180,E1 -14535.065,E2 -14535.065} C_VEL
LIN {X 0,Y 333.636,Z 185.928,A -85,B 0,C 180,E1 -14539.314,E2 -14539.314} C_VEL
LIN {X 0,Y 333.651,Z 185.925,A -85,B 0,C 180,E1 -14543.167,E2 -14543.167} C_VEL
LIN {X 0,Y 333.66,Z 185.926,A -85,B 0,C 180,E1 -14545.34,E2 -14545.34} C_VEL
LIN {X 0,Y 333.613,Z 185.927,A -85,B 0,C 180,E1 -14548.22,E2 -14548.22} C_VEL
LIN {X 0,Y 333.696,Z 185.916,A -85,B 0,C 180,E1 -14552.192,E2 -14552.192} C_VEL
LIN {X 0,Y 333.716,Z 185.918,A -85,B 0,C 180,E1 -14555.09,E2 -14555.09} C_VEL
LIN {X 0,Y 333.703,Z 185.92,A -85,B 0,C 180,E1 -14559.021,E2 -14559.021} C_VEL
LIN {X 0,Y 333.777,Z 185.906,A -85,B 0,C 180,E1 -14561.589,E2 -14561.589} C_VEL
LIN {X 0,Y 333.79,Z 185.904,A -85,B 0,C 180,E1 -14565.576,E2 -14565.576} C_VEL
LIN {X 0,Y 333.817,Z 185.902,A -85,B 0,C 180,E1 -14569.078,E2 -14569.078} C_VEL
LIN {X 0,Y 333.996,Z 185.881,A -85,B 0,C 180,E1 -14572.747,E2 -14572.747} C_VEL
LIN {X 0,Y 333.794,Z 185.903,A -85,B 0,C 180,E1 -14575.169,E2 -14575.169} C_VEL
LIN {X 0,Y 334.083,Z 185.868,A -85,B 0,C 180,E1 -14577.589,E2 -14577.589} C_VEL
LIN {X 0,Y 334.168,Z 185.86,A -85,B 0,C 180,E1 -14580,E2 -14580} C_VEL
LIN {X 0,Y 334.12,Z 185.866,A -85,B 0,C 180,E1 -14582.411,E2 -14582.411} C_VEL
LIN {X 0,Y 333.975,Z 185.881,A -85,B 0,C 180,E1 -14586.596,E2 -14586.596} C_VEL
LIN {X 0,Y 333.803,Z 185.906,A -85,B 0,C 180,E1 -14589.697,E2 -14589.697} C_VEL
LIN {X 0,Y 333.777,Z 185.908,A -85,B 0,C 180,E1 -14593.393,E2 -14593.393} C_VEL
LIN {X 0,Y 333.733,Z 185.912,A -85,B 0,C 180,E1 -14597.147,E2 -14597.147} C_VEL
LIN {X 0,Y 333.72,Z 185.917,A -85,B 0,C 180,E1 -14599.692,E2 -14599.692} C_VEL
LIN {X 0,Y 333.677,Z 185.918,A -85,B 0,C 180,E1 -14602.28,E2 -14602.28} C_VEL
LIN {X 0,Y 333.72,Z 185.912,A -85,B 0,C 180,E1 -14606.248,E2 -14606.248} C_VEL
LIN {X 0,Y 333.697,Z 185.918,A -85,B 0,C 180,E1 -14608.974,E2 -14608.974} C_VEL
LIN {X 0,Y 333.631,Z 185.925,A -85,B 0,C 180,E1 -14612.589,E2 -14612.589} C_VEL
LIN {X 0,Y 333.664,Z 185.92,A -85,B 0,C 180,E1 -14616.141,E2 -14616.141} C_VEL
LIN {X 0,Y 333.636,Z 185.926,A -85,B 0,C 180,E1 -14619.194,E2 -14619.194} C_VEL
LIN {X 0,Y 333.623,Z 185.927,A -85,B 0,C 180,E1 -14622.502,E2 -14622.502} C_VEL
LIN {X 0,Y 333.588,Z 185.93,A -85,B 0,C 180,E1 -14625.957,E2 -14625.957} C_VEL
LIN {X 0,Y 333.597,Z 185.931,A -85,B 0,C 180,E1 -14629.326,E2 -14629.326} C_VEL
LIN {X 0,Y 333.688,Z 186.928,A -85,B 0,C 180,E1 -14631.195,E2 -14631.195} C_VEL
LIN {X 0,Y 333.704,Z 189.569,A -85,B 0,C 180,E1 -14633.867,E2 -14633.867} C_VEL
LIN {X 0,Y 333.468,Z 192.569,A -85,B 0,C 180,E1 -14636.774,E2 -14636.774} C_VEL
LIN {X 0,Y 333.165,Z 197.122,A -85,B 0,C 180,E1 -14640.977,E2 -14640.977} C_VEL
LIN {X 0,Y 332.985,Z 200.151,A -85,B 0,C 180,E1 -14643.691,E2 -14643.691} C_VEL
LIN {X 0,Y 332.846,Z 202.545,A -85,B 0,C 180,E1 -14645.794,E2 -14645.794} C_VEL
LIN {X 0,Y 336.528,Z 215.543,A -85,B 0,C 180,E1 -14646.603,E2 -14646.603} C_VEL
LIN {X 0,Y 339.497,Z 228.233,A -85,B 0,C 180,E1 -14647.596,E2 -14647.596} C_VEL
LIN {X 0,Y 340.986,Z 237.375,A -85,B 0,C 180,E1 -14648.435,E2 -14648.435} C_VEL
LIN {X 0,Y 339.986,Z 247.9,A -85,B 0,C 180,E1 -14649.427,E2 -14649.427} C_VEL
LIN {X 0,Y 338.519,Z 259.209,A -85,B 0,C 180,E1 -14650.757,E2 -14650.757} C_VEL
LIN {X 0,Y 337.358,Z 268.292,A -85,B 0,C 180,E1 -14652.105,E2 -14652.105} C_VEL
LIN {X 0,Y 336.076,Z 276.603,A -85,B 0,C 180,E1 -14653.602,E2 -14653.602} C_VEL
LIN {X 0,Y 334.874,Z 284.723,A -85,B 0,C 180,E1 -14655.414,E2 -14655.414} C_VEL
LIN {X 0,Y 333.998,Z 291.245,A -85,B 0,C 180,E1 -14657.236,E2 -14657.236} C_VEL
LIN {X 0,Y 333.177,Z 296.431,A -85,B 0,C 180,E1 -14659.056,E2 -14659.056} C_VEL
LIN {X 0,Y 332.701,Z 300.45,A -85,B 0,C 180,E1 -14660.884,E2 -14660.884} C_VEL
LIN {X 0,Y 332.336,Z 303.421,A -85,B 0,C 180,E1 -14662.71,E2 -14662.71} C_VEL
LIN {X 0,Y 332.142,Z 304.934,A -85,B 0,C 180,E1 -14663.995,E2 -14663.995} C_VEL
LIN {X 0,Y 332.034,Z 306.524,A -85,B 0,C 180,E1 -14666.359,E2 -14666.359} C_VEL
LIN {X 0,Y 331.957,Z 306.781,A -85,B 0,C 180,E1 -14667.573,E2 -14667.573} C_VEL
LIN {X 0,Y 331.954,Z 306.636,A -85,B 0,C 180,E1 -14668.786,E2 -14668.786} C_VEL
LIN {X 0,Y 332.04,Z 305.129,A -85,B 0,C 180,E1 -14671.212,E2 -14671.212} C_VEL
LIN {X 0,Y 332.173,Z 303.797,A -85,B 0,C 180,E1 -14672.424,E2 -14672.424} C_VEL
LIN {X 0,Y 332.465,Z 300.98,A -85,B 0,C 180,E1 -14674.242,E2 -14674.242} C_VEL
LIN {X 0,Y 332.887,Z 297.152,A -85,B 0,C 180,E1 -14676.058,E2 -14676.058} C_VEL
LIN {X 0,Y 333.527,Z 291.369,A -85,B 0,C 180,E1 -14678.145,E2 -14678.145} C_VEL
LIN {X 0,Y 334.265,Z 284.791,A -85,B 0,C 180,E1 -14679.987,E2 -14679.987} C_VEL
LIN {X 0,Y 335.409,Z 276.73,A -85,B 0,C 180,E1 -14681.787,E2 -14681.787} C_VEL
LIN {X 0,Y 336.475,Z 268.496,A -85,B 0,C 180,E1 -14683.281,E2 -14683.281} C_VEL
LIN {X 0,Y 337.64,Z 258.406,A -85,B 0,C 180,E1 -14684.771,E2 -14684.771} C_VEL
LIN {X 0,Y 338.509,Z 249.805,A -85,B 0,C 180,E1 -14685.811,E2 -14685.811} C_VEL
LIN {X 0,Y 339.548,Z 239.259,A -85,B 0,C 180,E1 -14686.842,E2 -14686.842} C_VEL
LIN {X 0,Y 339.834,Z 235.801,A -85,B 0,C 180,E1 -14687.133,E2 -14687.133} C_VEL
LIN {X 0,Y 337.866,Z 223.273,A -85,B 0,C 180,E1 -14688.179,E2 -14688.179} C_VEL
LIN {X 0,Y 334.816,Z 210.454,A -85,B 0,C 180,E1 -14689.048,E2 -14689.048} C_VEL
LIN {X 0,Y 332.694,Z 202.452,A -85,B 0,C 180,E1 -14689.494,E2 -14689.494} C_VEL
LIN {X 0,Y 332.875,Z 199.173,A -85,B 0,C 180,E1 -14692.333,E2 -14692.333} C_VEL
LIN {X 0,Y 333.137,Z 194.692,A -85,B 0,C 180,E1 -14696.294,E2 -14696.294} C_VEL
LIN {X 0,Y 333.411,Z 190.418,A -85,B 0,C 180,E1 -14700.202,E2 -14700.202} C_VEL
LIN {X 0,Y 333.549,Z 187.286,A -85,B 0,C 180,E1 -14703.214,E2 -14703.214} C_VEL
LIN {X 0,Y 333.584,Z 185.934,A -85,B 0,C 180,E1 -14704.748,E2 -14704.748} C_VEL
LIN {X 0,Y 333.637,Z 185.928,A -85,B 0,C 180,E1 -14707.649,E2 -14707.649} C_VEL
LIN {X 0,Y 333.635,Z 185.924,A -85,B 0,C 180,E1 -14710.764,E2 -14710.764} C_VEL
LIN {X 0,Y 333.629,Z 185.924,A -85,B 0,C 180,E1 -14714.256,E2 -14714.256} C_VEL
LIN {X 0,Y 333.678,Z 185.919,A -85,B 0,C 180,E1 -14717.624,E2 -14717.624} C_VEL
LIN {X 0,Y 333.662,Z 185.924,A -85,B 0,C 180,E1 -14721.194,E2 -14721.194} C_VEL
LIN {X 0,Y 333.654,Z 185.922,A -85,B 0,C 180,E1 -14725.047,E2 -14725.047} C_VEL
LIN {X 0,Y 333.044,Z 186.005,A -85,B 0,C 180,E1 -14726.053,E2 -14726.053} C_VEL
LIN {X 0,Y 330.24,Z 186.361,A -85,B 0,C 180,E1 -14727.691,E2 -14727.691} C_VEL
LIN {X 0,Y 327.812,Z 186.66,A -85,B 0,C 180,E1 -14729.017,E2 -14729.017} C_VEL
LIN {X 0,Y 326.738,Z 186.787,A -85,B 0,C 180,E1 -14730.044,E2 -14730.044} C_VEL
LIN {X 0,Y 326.635,Z 186.797,A -85,B 0,C 180,E1 -14730.391,E2 -14730.391} C_VEL
LIN {X 0,Y 326.669,Z 186.796,A -85,B 0,C 180,E1 -14734.514,E2 -14734.514} C_VEL
LIN {X 0,Y 326.644,Z 186.79,A -85,B 0,C 180,E1 -14738.545,E2 -14738.545} C_VEL
LIN {X 0,Y 326.72,Z 186.781,A -85,B 0,C 180,E1 -14741.176,E2 -14741.176} C_VEL
LIN {X 0,Y 326.737,Z 186.783,A -85,B 0,C 180,E1 -14745.432,E2 -14745.432} C_VEL
LIN {X 0,Y 326.753,Z 186.778,A -85,B 0,C 180,E1 -14748.838,E2 -14748.838} C_VEL
LIN {X 0,Y 326.946,Z 186.756,A -85,B 0,C 180,E1 -14751.388,E2 -14751.388} C_VEL
LIN {X 0,Y 326.976,Z 186.757,A -85,B 0,C 180,E1 -14753.83,E2 -14753.83} C_VEL
LIN {X 0,Y 327.018,Z 186.748,A -85,B 0,C 180,E1 -14757.536,E2 -14757.536} C_VEL
LIN {X 0,Y 327.13,Z 186.737,A -85,B 0,C 180,E1 -14760,E2 -14760} C_VEL
LIN {X 0,Y 327.048,Z 186.744,A -85,B 0,C 180,E1 -14762.463,E2 -14762.463} C_VEL
LIN {X 0,Y 326.971,Z 186.754,A -85,B 0,C 180,E1 -14766.169,E2 -14766.169} C_VEL
LIN {X 0,Y 326.887,Z 186.764,A -85,B 0,C 180,E1 -14768.656,E2 -14768.656} C_VEL
LIN {X 0,Y 326.71,Z 186.786,A -85,B 0,C 180,E1 -14772.422,E2 -14772.422} C_VEL
LIN {X 0,Y 326.724,Z 186.787,A -85,B 0,C 180,E1 -14774.959,E2 -14774.959} C_VEL
LIN {X 0,Y 326.711,Z 186.789,A -85,B 0,C 180,E1 -14778.841,E2 -14778.841} C_VEL
LIN {X 0,Y 326.63,Z 186.799,A -85,B 0,C 180,E1 -14782.786,E2 -14782.786} C_VEL
LIN {X 0,Y 326.668,Z 186.792,A -85,B 0,C 180,E1 -14785.485,E2 -14785.485} C_VEL
LIN {X 0,Y 326.638,Z 186.793,A -85,B 0,C 180,E1 -14789.661,E2 -14789.661} C_VEL
LIN {X 0,Y 326.585,Z 186.802,A -85,B 0,C 180,E1 -14794.022,E2 -14794.022} C_VEL
LIN {X 0,Y 326.608,Z 186.799,A -85,B 0,C 180,E1 -14797.241,E2 -14797.241} C_VEL
LIN {X 0,Y 326.617,Z 186.801,A -85,B 0,C 180,E1 -14800.205,E2 -14800.205} C_VEL
LIN {X 0,Y 326.641,Z 186.796,A -85,B 0,C 180,E1 -14803.512,E2 -14803.512} C_VEL
LIN {X 0,Y 326.726,Z 186.959,A -85,B 0,C 180,E1 -14806.202,E2 -14806.202} C_VEL
LIN {X 0,Y 327.481,Z 191.621,A -85,B 0,C 180,E1 -14809.927,E2 -14809.927} C_VEL
LIN {X 0,Y 327.93,Z 194.986,A -85,B 0,C 180,E1 -14812.463,E2 -14812.463} C_VEL
LIN {X 0,Y 328.038,Z 198.055,A -85,B 0,C 180,E1 -14814.662,E2 -14814.662} C_VEL
LIN {X 0,Y 327.425,Z 203.37,A -85,B 0,C 180,E1 -14818.276,E2 -14818.276} C_VEL
LIN {X 0,Y 326.769,Z 208.811,A -85,B 0,C 180,E1 -14821.862,E2 -14821.862} C_VEL
LIN {X 0,Y 326.138,Z 214.984,A -85,B 0,C 180,E1 -14825.833,E2 -14825.833} C_VEL
LIN {X 0,Y 325.897,Z 218.493,A -85,B 0,C 180,E1 -14828.067,E2 -14828.067} C_VEL
LIN {X 0,Y 328.805,Z 232.771,A -85,B 0,C 180,E1 -14828.847,E2 -14828.847} C_VEL
LIN {X 0,Y 330.78,Z 246.062,A -85,B 0,C 180,E1 -14829.796,E2 -14829.796} C_VEL
LIN {X 0,Y 331.915,Z 257.772,A -85,B 0,C 180,E1 -14830.843,E2 -14830.843} C_VEL
LIN {X 0,Y 330.947,Z 268.23,A -85,B 0,C 180,E1 -14831.908,E2 -14831.908} C_VEL
LIN {X 0,Y 329.595,Z 278.996,A -85,B 0,C 180,E1 -14833.272,E2 -14833.272} C_VEL
LIN {X 0,Y 328.41,Z 289.101,A -85,B 0,C 180,E1 -14834.876,E2 -14834.876} C_VEL
LIN {X 0,Y 327.254,Z 298.043,A -85,B 0,C 180,E1 -14836.654,E2 -14836.654} C_VEL
LIN {X 0,Y 326.24,Z 305.529,A -85,B 0,C 180,E1 -14838.508,E2 -14838.508} C_VEL
LIN {X 0,Y 325.551,Z 312.447,A -85,B 0,C 180,E1 -14840.684,E2 -14840.684} C_VEL
LIN {X 0,Y 325.174,Z 317.007,A -85,B 0,C 180,E1 -14842.55,E2 -14842.55} C_VEL
LIN {X 0,Y 324.924,Z 320.194,A -85,B 0,C 180,E1 -14844.249,E2 -14844.249} C_VEL
LIN {X 0,Y 324.9,Z 322.935,A -85,B 0,C 180,E1 -14846.28,E2 -14846.28} C_VEL
LIN {X 0,Y 324.836,Z 324.042,A -85,B 0,C 180,E1 -14847.521,E2 -14847.521} C_VEL
LIN {X 0,Y 324.873,Z 325.051,A -85,B 0,C 180,E1 -14850.001,E2 -14850.001} C_VEL
LIN {X 0,Y 324.821,Z 324.975,A -85,B 0,C 180,E1 -14851.241,E2 -14851.241} C_VEL
LIN {X 0,Y 324.834,Z 324.482,A -85,B 0,C 180,E1 -14852.481,E2 -14852.481} C_VEL
LIN {X 0,Y 324.874,Z 323.574,A -85,B 0,C 180,E1 -14853.722,E2 -14853.722} C_VEL
LIN {X 0,Y 324.959,Z 320.565,A -85,B 0,C 180,E1 -14856.208,E2 -14856.208} C_VEL
LIN {X 0,Y 325.286,Z 317.139,A -85,B 0,C 180,E1 -14858.073,E2 -14858.073} C_VEL
LIN {X 0,Y 325.79,Z 312.641,A -85,B 0,C 180,E1 -14859.938,E2 -14859.938} C_VEL
LIN {X 0,Y 326.649,Z 305.835,A -85,B 0,C 180,E1 -14862.109,E2 -14862.109} C_VEL
LIN {X 0,Y 327.844,Z 298.448,A -85,B 0,C 180,E1 -14863.955,E2 -14863.955} C_VEL
LIN {X 0,Y 329.138,Z 289.279,A -85,B 0,C 180,E1 -14865.798,E2 -14865.798} C_VEL
LIN {X 0,Y 330.453,Z 279.754,A -85,B 0,C 180,E1 -14867.322,E2 -14867.322} C_VEL
LIN {X 0,Y 331.938,Z 269.203,A -85,B 0,C 180,E1 -14868.677,E2 -14868.677} C_VEL
LIN {X 0,Y 333.05,Z 260.624,A -85,B 0,C 180,E1 -14869.572,E2 -14869.572} C_VEL
LIN {X 0,Y 332.222,Z 250.023,A -85,B 0,C 180,E1 -14870.597,E2 -14870.597} C_VEL
LIN {X 0,Y 330.545,Z 238.825,A -85,B 0,C 180,E1 -14871.515,E2 -14871.515} C_VEL
LIN {X 0,Y 327.848,Z 225.759,A -85,B 0,C 180,E1 -14872.391,E2 -14872.391} C_VEL
LIN {X 0,Y 326.111,Z 218.316,A -85,B 0,C 180,E1 -14872.824,E2 -14872.824} C_VEL
LIN {X 0,Y 326.676,Z 212.083,A -85,B 0,C 180,E1 -14876.857,E2 -14876.857} C_VEL
LIN {X 0,Y 327.45,Z 206.07,A -85,B 0,C 180,E1 -14880.85,E2 -14880.85} C_VEL
LIN {X 0,Y 328.124,Z 200.639,A -85,B 0,C 180,E1 -14884.581,E2 -14884.581} C_VEL
LIN {X 0,Y 328.123,Z 196.49,A -85,B 0,C 180,E1 -14887.581,E2 -14887.581} C_VEL
LIN {X 0,Y 327.738,Z 193.321,A -85,B 0,C 180,E1 -14890.037,E2 -14890.037} C_VEL
LIN {X 0,Y 327.068,Z 189.153,A -85,B 0,C 180,E1 -14893.439,E2 -14893.439} C_VEL
LIN {X 0,Y 326.606,Z 186.806,A -85,B 0,C 180,E1 -14895.528,E2 -14895.528} C_VEL
LIN {X 0,Y 326.58,Z 186.806,A -85,B 0,C 180,E1 -14899.789,E2 -14899.789} C_VEL
LIN {X 0,Y 326.617,Z 186.8,A -85,B 0,C 180,E1 -14902.951,E2 -14902.951} C_VEL
LIN {X 0,Y 326.593,Z 186.802,A -85,B 0,C 180,E1 -14905.979,E2 -14905.979} C_VEL
LIN {X 0,Y 326.598,Z 186.805,A -85,B 0,C 180,E1 -14909.396,E2 -14909.396} C_VEL
LIN {X 0,Y 326.662,Z 186.797,A -85,B 0,C 180,E1 -14913.141,E2 -14913.141} C_VEL
LIN {X 0,Y 326.647,Z 186.794,A -85,B 0,C 180,E1 -14915.871,E2 -14915.871} C_VEL
LIN {X 0,Y 326.669,Z 186.791,A -85,B 0,C 180,E1 -14919.866,E2 -14919.866} C_VEL
LIN {X 0,Y 326.682,Z 186.792,A -85,B 0,C 180,E1 -14922.471,E2 -14922.471} C_VEL
LIN {X 0,Y 326.739,Z 186.785,A -85,B 0,C 180,E1 -14926.314,E2 -14926.314} C_VEL
LIN {X 0,Y 326.795,Z 186.777,A -85,B 0,C 180,E1 -14930.093,E2 -14930.093} C_VEL
LIN {X 0,Y 326.979,Z 186.753,A -85,B 0,C 180,E1 -14933.831,E2 -14933.831} C_VEL
LIN {X 0,Y 327.025,Z 186.747,A -85,B 0,C 180,E1 -14937.537,E2 -14937.537} C_VEL
LIN {X 0,Y 327.121,Z 186.738,A -85,B 0,C 180,E1 -14940,E2 -14940} C_VEL
LIN {X 0,Y 327.057,Z 186.745,A -85,B 0,C 180,E1 -14942.463,E2 -14942.463} C_VEL
LIN {X 0,Y 326.943,Z 186.758,A -85,B 0,C 180,E1 -14946.586,E2 -14946.586} C_VEL
LIN {X 0,Y 326.765,Z 186.784,A -85,B 0,C 180,E1 -14949.908,E2 -14949.908} C_VEL
LIN {X 0,Y 326.74,Z 186.787,A -85,B 0,C 180,E1 -14953.687,E2 -14953.687} C_VEL
LIN {X 0,Y 326.685,Z 186.794,A -85,B 0,C 180,E1 -14957.529,E2 -14957.529} C_VEL
LIN {X 0,Y 326.646,Z 186.795,A -85,B 0,C 180,E1 -14960.136,E2 -14960.136} C_VEL
LIN {X 0,Y 326.636,Z 186.795,A -85,B 0,C 180,E1 -14964.131,E2 -14964.131} C_VEL
LIN {X 0,Y 326.67,Z 186.792,A -85,B 0,C 180,E1 -14966.859,E2 -14966.859} C_VEL
LIN {X 0,Y 326.626,Z 186.797,A -85,B 0,C 180,E1 -14970.613,E2 -14970.613} C_VEL
LIN {X 0,Y 326.595,Z 186.8,A -85,B 0,C 180,E1 -14974.021,E2 -14974.021} C_VEL
LIN {X 0,Y 326.616,Z 186.801,A -85,B 0,C 180,E1 -14977.24,E2 -14977.24} C_VEL
LIN {X 0,Y 326.569,Z 186.806,A -85,B 0,C 180,E1 -14981.133,E2 -14981.133} C_VEL
LIN {X 0,Y 326.519,Z 186.815,A -85,B 0,C 180,E1 -14984.744,E2 -14984.744} C_VEL
LIN {X 0,Y 326.557,Z 186.808,A -85,B 0,C 180,E1 -14988.154,E2 -14988.154} C_VEL
LIN {X 0,Y 326.542,Z 186.81,A -85,B 0,C 180,E1 -14989.786,E2 -14989.786} C_VEL
LIN {X 0,Y 326.72,Z 189.472,A -85,B 0,C 180,E1 -14992.741,E2 -14992.741} C_VEL
LIN {X 0,Y 326.512,Z 192.708,A -85,B 0,C 180,E1 -14995.971,E2 -14995.971} C_VEL
LIN {X 0,Y 326.228,Z 196.455,A -85,B 0,C 180,E1 -14999.512,E2 -14999.512} C_VEL
LIN {X 0,Y 325.951,Z 200.312,A -85,B 0,C 180,E1 -15003.078,E2 -15003.078} C_VEL
LIN {X 0,Y 325.826,Z 202.946,A -85,B 0,C 180,E1 -15005.272,E2 -15005.272} C_VEL
LIN {X 0,Y 329.708,Z 216.269,A -85,B 0,C 180,E1 -15006.145,E2 -15006.145} C_VEL
LIN {X 0,Y 332.45,Z 227.871,A -85,B 0,C 180,E1 -15007.08,E2 -15007.08} C_VEL
LIN {X 0,Y 334.154,Z 237.872,A -85,B 0,C 180,E1 -15008.024,E2 -15008.024} C_VEL
LIN {X 0,Y 333.337,Z 247.876,A -85,B 0,C 180,E1 -15008.997,E2 -15008.997} C_VEL
LIN {X 0,Y 331.806,Z 259.234,A -85,B 0,C 180,E1 -15010.352,E2 -15010.352} C_VEL
LIN {X 0,Y 330.566,Z 268.351,A -85,B 0,C 180,E1 -15011.725,E2 -15011.725} C_VEL
LIN {X 0,Y 329.226,Z 276.686,A -85,B 0,C 180,E1 -15013.251,E2 -15013.251} C_VEL
LIN {X 0,Y 327.943,Z 284.826,A -85,B 0,C 180,E1 -15015.098,E2 -15015.098} C_VEL
LIN {X 0,Y 327.068,Z 291.365,A -85,B 0,C 180,E1 -15016.961,E2 -15016.961} C_VEL
LIN {X 0,Y 326.18,Z 296.566,A -85,B 0,C 180,E1 -15018.818,E2 -15018.818} C_VEL
LIN {X 0,Y 325.662,Z 300.6,A -85,B 0,C 180,E1 -15020.685,E2 -15020.685} C_VEL
LIN {X 0,Y 325.279,Z 303.584,A -85,B 0,C 180,E1 -15022.551,E2 -15022.551} C_VEL
LIN {X 0,Y 325.045,Z 305.274,A -85,B 0,C 180,E1 -15024.046,E2 -15024.046} C_VEL
LIN {X 0,Y 324.964,Z 306.712,A -85,B 0,C 180,E1 -15026.279,E2 -15026.279} C_VEL
LIN {X 0,Y 324.875,Z 306.975,A -85,B 0,C 180,E1 -15027.52,E2 -15027.52} C_VEL
LIN {X 0,Y 324.861,Z 306.842,A -85,B 0,C 180,E1 -15028.76,E2 -15028.76} C_VEL
LIN {X 0,Y 324.947,Z 305.349,A -85,B 0,C 180,E1 -15031.238,E2 -15031.238} C_VEL
LIN {X 0,Y 325.086,Z 304.023,A -85,B 0,C 180,E1 -15032.477,E2 -15032.477} C_VEL
LIN {X 0,Y 325.397,Z 301.219,A -85,B 0,C 180,E1 -15034.334,E2 -15034.334} C_VEL
LIN {X 0,Y 325.836,Z 297.405,A -85,B 0,C 180,E1 -15036.19,E2 -15036.19} C_VEL
LIN {X 0,Y 326.472,Z 291.883,A -85,B 0,C 180,E1 -15038.245,E2 -15038.245} C_VEL
LIN {X 0,Y 327.293,Z 285.085,A -85,B 0,C 180,E1 -15040.202,E2 -15040.202} C_VEL
LIN {X 0,Y 328.487,Z 277.042,A -85,B 0,C 180,E1 -15042.039,E2 -15042.039} C_VEL
LIN {X 0,Y 329.584,Z 268.832,A -85,B 0,C 180,E1 -15043.564,E2 -15043.564} C_VEL
LIN {X 0,Y 330.806,Z 258.785,A -85,B 0,C 180,E1 -15045.083,E2 -15045.083} C_VEL
LIN {X 0,Y 331.719,Z 250.209,A -85,B 0,C 180,E1 -15046.143,E2 -15046.143} C_VEL
LIN {X 0,Y 332.697,Z 241.347,A -85,B 0,C 180,E1 -15047.042,E2 -15047.042} C_VEL
LIN {X 0,Y 332.893,Z 235.61,A -85,B 0,C 180,E1 -15047.563,E2 -15047.563} C_VEL
LIN {X 0,Y 330.99,Z 223.888,A -85,B 0,C 180,E1 -15048.57,E2 -15048.57} C_VEL
LIN {X 0,Y 327.977,Z 211.19,A -85,B 0,C 180,E1 -15049.463,E2 -15049.463} C_VEL
LIN {X 0,Y 325.647,Z 202.662,A -85,B 0,C 180,E1 -15049.959,E2 -15049.959} C_VEL
LIN {X 0,Y 325.841,Z 199.379,A -85,B 0,C 180,E1 -15052.842,E2 -15052.842} C_VEL
LIN {X 0,Y 326.041,Z 196.394,A -85,B 0,C 180,E1 -15055.535,E2 -15055.535} C_VEL
LIN {X 0,Y 326.232,Z 193.386,A -85,B 0,C 180,E1 -15058.288,E2 -15058.288} C_VEL
LIN {X 0,Y 326.427,Z 190.417,A -85,B 0,C 180,E1 -15061.109,E2 -15061.109} C_VEL
LIN {X 0,Y 326.519,Z 187.48,A -85,B 0,C 180,E1 -15064.026,E2 -15064.026} C_VEL
LIN {X 0,Y 326.562,Z 186.81,A -85,B 0,C 180,E1 -15065.522,E2 -15065.522} C_VEL
LIN {X 0,Y 326.586,Z 186.803,A -85,B 0,C 180,E1 -15068.609,E2 -15068.609} C_VEL
LIN {X 0,Y 326.565,Z 186.806,A -85,B 0,C 180,E1 -15071.843,E2 -15071.843} C_VEL
LIN {X 0,Y 326.577,Z 186.807,A -85,B 0,C 180,E1 -15075.243,E2 -15075.243} C_VEL
LIN {X 0,Y 326.614,Z 186.801,A -85,B 0,C 180,E1 -15078.855,E2 -15078.855} C_VEL
LIN {X 0,Y 326.627,Z 186.798,A -85,B 0,C 180,E1 -15081.391,E2 -15081.391} C_VEL
LIN {X 0,Y 326.589,Z 186.804,A -85,B 0,C 180,E1 -15085.037,E2 -15085.037} C_VEL
LIN {X 0,Y 326.587,Z 186.801,A -85,B 0,C 180,E1 -15087.453,E2 -15087.453} C_VEL
LIN {X 0,Y 326.635,Z 186.797,A -85,B 0,C 180,E1 -15090.391,E2 -15090.391} C_VEL
LIN {X 0,Y 325.928,Z 186.884,A -85,B 0,C 180,E1 -15091.421,E2 -15091.421} C_VEL
LIN {X 0,Y 323.071,Z 187.241,A -85,B 0,C 180,E1 -15093.098,E2 -15093.098} C_VEL
LIN {X 0,Y 320.676,Z 187.542,A -85,B 0,C 180,E1 -15094.456,E2 -15094.456} C_VEL
LIN {X 0,Y 319.651,Z 187.663,A -85,B 0,C 180,E1 -15095.508,E2 -15095.508} C_VEL
LIN {X 0,Y 319.568,Z 187.671,A -85,B 0,C 180,E1 -15095.864,E2 -15095.864} C_VEL
LIN {X 0,Y 319.609,Z 187.66,A -85,B 0,C 180,E1 -15099.4,E2 -15099.4} C_VEL
LIN {X 0,Y 319.634,Z 187.665,A -85,B 0,C 180,E1 -15102.071,E2 -15102.071} C_VEL
LIN {X 0,Y 319.707,Z 187.662,A -85,B 0,C 180,E1 -15106.006,E2 -15106.006} C_VEL
LIN {X 0,Y 319.756,Z 187.653,A -85,B 0,C 180,E1 -15109.872,E2 -15109.872} C_VEL
LIN {X 0,Y 319.92,Z 187.633,A -85,B 0,C 180,E1 -15112.426,E2 -15112.426} C_VEL
LIN {X 0,Y 319.725,Z 187.655,A -85,B 0,C 180,E1 -15114.955,E2 -15114.955} C_VEL
LIN {X 0,Y 319.962,Z 187.626,A -85,B 0,C 180,E1 -15117.482,E2 -15117.482} C_VEL
LIN {X 0,Y 320.083,Z 187.615,A -85,B 0,C 180,E1 -15120,E2 -15120} C_VEL
LIN {X 0,Y 319.989,Z 187.623,A -85,B 0,C 180,E1 -15122.517,E2 -15122.517} C_VEL
LIN {X 0,Y 319.926,Z 187.631,A -85,B 0,C 180,E1 -15126.306,E2 -15126.306} C_VEL
LIN {X 0,Y 319.816,Z 187.646,A -85,B 0,C 180,E1 -15128.848,E2 -15128.848} C_VEL
LIN {X 0,Y 319.656,Z 187.665,A -85,B 0,C 180,E1 -15132.701,E2 -15132.701} C_VEL
LIN {X 0,Y 319.655,Z 187.67,A -85,B 0,C 180,E1 -15135.298,E2 -15135.298} C_VEL
LIN {X 0,Y 319.655,Z 187.67,A -85,B 0,C 180,E1 -15139.256,E2 -15139.256} C_VEL
LIN {X 0,Y 319.59,Z 187.676,A -85,B 0,C 180,E1 -15143.318,E2 -15143.318} C_VEL
LIN {X 0,Y 319.612,Z 187.67,A -85,B 0,C 180,E1 -15146.09,E2 -15146.09} C_VEL
LIN {X 0,Y 319.567,Z 187.678,A -85,B 0,C 180,E1 -15148.936,E2 -15148.936} C_VEL
LIN {X 0,Y 319.51,Z 187.681,A -85,B 0,C 180,E1 -15151.864,E2 -15151.864} C_VEL
LIN {X 0,Y 319.559,Z 187.677,A -85,B 0,C 180,E1 -15155.545,E2 -15155.545} C_VEL
LIN {X 0,Y 319.563,Z 187.678,A -85,B 0,C 180,E1 -15158.009,E2 -15158.009} C_VEL
LIN {X 0,Y 319.584,Z 187.675,A -85,B 0,C 180,E1 -15161.615,E2 -15161.615} C_VEL
LIN {X 0,Y 319.632,Z 187.673,A -85,B 0,C 180,E1 -15165.288,E2 -15165.288} C_VEL
LIN {X 0,Y 319.652,Z 187.823,A -85,B 0,C 180,E1 -15165.841,E2 -15165.841} C_VEL
LIN {X 0,Y 320.253,Z 191.429,A -85,B 0,C 180,E1 -15168.83,E2 -15168.83} C_VEL
LIN {X 0,Y 320.88,Z 195.718,A -85,B 0,C 180,E1 -15172.179,E2 -15172.179} C_VEL
LIN {X 0,Y 320.994,Z 198.314,A -85,B 0,C 180,E1 -15174.105,E2 -15174.105} C_VEL
LIN {X 0,Y 320.644,Z 202.105,A -85,B 0,C 180,E1 -15176.777,E2 -15176.777} C_VEL
LIN {X 0,Y 319.981,Z 207.399,A -85,B 0,C 180,E1 -15180.387,E2 -15180.387} C_VEL
LIN {X 0,Y 319.266,Z 213.581,A -85,B 0,C 180,E1 -15184.493,E2 -15184.493} C_VEL
LIN {X 0,Y 318.863,Z 218.299,A -85,B 0,C 180,E1 -15187.589,E2 -15187.589} C_VEL
LIN {X 0,Y 321.689,Z 231.816,A -85,B 0,C 180,E1 -15188.337,E2 -15188.337} C_VEL
LIN {X 0,Y 323.624,Z 244.171,A -85,B 0,C 180,E1 -15189.228,E2 -15189.228} C_VEL
LIN {X 0,Y 324.839,Z 255.573,A -85,B 0,C 180,E1 -15190.244,E2 -15190.244} C_VEL
LIN {X 0,Y 325.02,Z 260.579,A -85,B 0,C 180,E1 -15190.748,E2 -15190.748} C_VEL
LIN {X 0,Y 323.685,Z 271.764,A -85,B 0,C 180,E1 -15191.979,E2 -15191.979} C_VEL
LIN {X 0,Y 322.516,Z 280.816,A -85,B 0,C 180,E1 -15193.22,E2 -15193.22} C_VEL
LIN {X 0,Y 321.346,Z 290.106,A -85,B 0,C 180,E1 -15194.787,E2 -15194.787} C_VEL
LIN {X 0,Y 320.117,Z 299.124,A -85,B 0,C 180,E1 -15196.674,E2 -15196.674} C_VEL
LIN {X 0,Y 319.112,Z 306.386,A -85,B 0,C 180,E1 -15198.569,E2 -15198.569} C_VEL
LIN {X 0,Y 318.499,Z 312.197,A -85,B 0,C 180,E1 -15200.476,E2 -15200.476} C_VEL
LIN {X 0,Y 318.093,Z 316.769,A -85,B 0,C 180,E1 -15202.384,E2 -15202.384} C_VEL
LIN {X 0,Y 317.835,Z 320.25,A -85,B 0,C 180,E1 -15204.294,E2 -15204.294} C_VEL
LIN {X 0,Y 317.808,Z 322.715,A -85,B 0,C 180,E1 -15206.197,E2 -15206.197} C_VEL
LIN {X 0,Y 317.758,Z 323.833,A -85,B 0,C 180,E1 -15207.466,E2 -15207.466} C_VEL
LIN {X 0,Y 317.78,Z 324.851,A -85,B 0,C 180,E1 -15210.001,E2 -15210.001} C_VEL
LIN {X 0,Y 317.733,Z 324.78,A -85,B 0,C 180,E1 -15211.268,E2 -15211.268} C_VEL
LIN {X 0,Y 317.755,Z 324.296,A -85,B 0,C 180,E1 -15212.536,E2 -15212.536} C_VEL
LIN {X 0,Y 317.783,Z 323.392,A -85,B 0,C 180,E1 -15213.805,E2 -15213.805} C_VEL
LIN {X 0,Y 317.889,Z 320.393,A -85,B 0,C 180,E1 -15216.347,E2 -15216.347} C_VEL
LIN {X 0,Y 318.229,Z 316.978,A -85,B 0,C 180,E1 -15218.254,E2 -15218.254} C_VEL
LIN {X 0,Y 318.769,Z 312.491,A -85,B 0,C 180,E1 -15220.159,E2 -15220.159} C_VEL
LIN {X 0,Y 319.689,Z 305.703,A -85,B 0,C 180,E1 -15222.377,E2 -15222.377} C_VEL
LIN {X 0,Y 320.948,Z 298.331,A -85,B 0,C 180,E1 -15224.261,E2 -15224.261} C_VEL
LIN {X 0,Y 322.171,Z 289.974,A -85,B 0,C 180,E1 -15225.994,E2 -15225.994} C_VEL
LIN {X 0,Y 323.508,Z 280.857,A -85,B 0,C 180,E1 -15227.526,E2 -15227.526} C_VEL
LIN {X 0,Y 325.011,Z 270.452,A -85,B 0,C 180,E1 -15228.926,E2 -15228.926} C_VEL
LIN {X 0,Y 326.287,Z 260.617,A -85,B 0,C 180,E1 -15229.994,E2 -15229.994} C_VEL
LIN {X 0,Y 325.266,Z 249.346,A -85,B 0,C 180,E1 -15231.118,E2 -15231.118} C_VEL
LIN {X 0,Y 323.319,Z 236.812,A -85,B 0,C 180,E1 -15232.16,E2 -15232.16} C_VEL
LIN {X 0,Y 320.528,Z 224.053,A -85,B 0,C 180,E1 -15233.013,E2 -15233.013} C_VEL
LIN {X 0,Y 319.075,Z 218.148,A -85,B 0,C 180,E1 -15233.357,E2 -15233.357} C_VEL
LIN {X 0,Y 319.717,Z 211.907,A -85,B 0,C 180,E1 -15237.491,E2 -15237.491} C_VEL
LIN {X 0,Y 320.487,Z 206.475,A -85,B 0,C 180,E1 -15241.214,E2 -15241.214} C_VEL
LIN {X 0,Y 321.109,Z 201.562,A -85,B 0,C 180,E1 -15244.682,E2 -15244.682} C_VEL
LIN {X 0,Y 321.088,Z 197.369,A -85,B 0,C 180,E1 -15247.795,E2 -15247.795} C_VEL
LIN {X 0,Y 320.565,Z 193.193,A -85,B 0,C 180,E1 -15251.123,E2 -15251.123} C_VEL
LIN {X 0,Y 319.892,Z 189.063,A -85,B 0,C 180,E1 -15254.668,E2 -15254.668} C_VEL
LIN {X 0,Y 319.558,Z 187.684,A -85,B 0,C 180,E1 -15255.96,E2 -15255.96} C_VEL
LIN {X 0,Y 319.548,Z 187.679,A -85,B 0,C 180,E1 -15260.33,E2 -15260.33} C_VEL
LIN {X 0,Y 319.566,Z 187.678,A -85,B 0,C 180,E1 -15264.456,E2 -15264.456} C_VEL
LIN {X 0,Y 319.509,Z 187.685,A -85,B 0,C 180,E1 -15268.136,E2 -15268.136} C_VEL
LIN {X 0,Y 319.594,Z 187.675,A -85,B 0,C 180,E1 -15271.59,E2 -15271.59} C_VEL
LIN {X 0,Y 319.596,Z 187.675,A -85,B 0,C 180,E1 -15275.303,E2 -15275.303} C_VEL
LIN {X 0,Y 319.6,Z 187.672,A -85,B 0,C 180,E1 -15278.048,E2 -15278.048} C_VEL
LIN {X 0,Y 319.675,Z 187.667,A -85,B 0,C 180,E1 -15280.96,E2 -15280.96} C_VEL
LIN {X 0,Y 319.713,Z 187.658,A -85,B 0,C 180,E1 -15285.276,E2 -15285.276} C_VEL
LIN {X 0,Y 319.74,Z 187.655,A -85,B 0,C 180,E1 -15289.873,E2 -15289.873} C_VEL
LIN {X 0,Y 319.899,Z 187.639,A -85,B 0,C 180,E1 -15292.426,E2 -15292.426} C_VEL
LIN {X 0,Y 319.731,Z 187.656,A -85,B 0,C 180,E1 -15294.956,E2 -15294.956} C_VEL
LIN {X 0,Y 319.969,Z 187.626,A -85,B 0,C 180,E1 -15297.483,E2 -15297.483} C_VEL
LIN {X 0,Y 320.076,Z 187.616,A -85,B 0,C 180,E1 -15300,E2 -15300} C_VEL
LIN {X 0,Y 319.998,Z 187.624,A -85,B 0,C 180,E1 -15302.518,E2 -15302.518} C_VEL
LIN {X 0,Y 319.906,Z 187.634,A -85,B 0,C 180,E1 -15306.572,E2 -15306.572} C_VEL
LIN {X 0,Y 319.717,Z 187.66,A -85,B 0,C 180,E1 -15310.129,E2 -15310.129} C_VEL
LIN {X 0,Y 319.714,Z 187.657,A -85,B 0,C 180,E1 -15314.725,E2 -15314.725} C_VEL
LIN {X 0,Y 319.674,Z 187.664,A -85,B 0,C 180,E1 -15319.039,E2 -15319.039} C_VEL
LIN {X 0,Y 319.555,Z 187.681,A -85,B 0,C 180,E1 -15323.321,E2 -15323.321} C_VEL
LIN {X 0,Y 319.605,Z 187.671,A -85,B 0,C 180,E1 -15326.091,E2 -15326.091} C_VEL
LIN {X 0,Y 319.576,Z 187.677,A -85,B 0,C 180,E1 -15328.935,E2 -15328.935} C_VEL
LIN {X 0,Y 319.52,Z 187.682,A -85,B 0,C 180,E1 -15331.864,E2 -15331.864} C_VEL
LIN {X 0,Y 319.568,Z 187.677,A -85,B 0,C 180,E1 -15335.544,E2 -15335.544} C_VEL
LIN {X 0,Y 319.55,Z 187.678,A -85,B 0,C 180,E1 -15339.671,E2 -15339.671} C_VEL
LIN {X 0,Y 319.513,Z 187.684,A -85,B 0,C 180,E1 -15343.462,E2 -15343.462} C_VEL
LIN {X 0,Y 319.546,Z 187.683,A -85,B 0,C 180,E1 -15347.018,E2 -15347.018} C_VEL
LIN {X 0,Y 319.494,Z 187.69,A -85,B 0,C 180,E1 -15348.709,E2 -15348.709} C_VEL
LIN {X 0,Y 319.578,Z 188.333,A -85,B 0,C 180,E1 -15350.378,E2 -15350.378} C_VEL
LIN {X 0,Y 319.649,Z 191.332,A -85,B 0,C 180,E1 -15353.586,E2 -15353.586} C_VEL
LIN {X 0,Y 319.421,Z 194.474,A -85,B 0,C 180,E1 -15356.73,E2 -15356.73} C_VEL
LIN {X 0,Y 319.197,Z 197.435,A -85,B 0,C 180,E1 -15359.577,E2 -15359.577} C_VEL
LIN {X 0,Y 318.829,Z 202.003,A -85,B 0,C 180,E1 -15363.842,E2 -15363.842} C_VEL
LIN {X 0,Y 318.797,Z 202.945,A -85,B 0,C 180,E1 -15364.71,E2 -15364.71} C_VEL
LIN {X 0,Y 322.731,Z 216.372,A -85,B 0,C 180,E1 -15365.618,E2 -15365.618} C_VEL
LIN {X 0,Y 325.722,Z 228.917,A -85,B 0,C 180,E1 -15366.668,E2 -15366.668} C_VEL
LIN {X 0,Y 327.483,Z 239.559,A -85,B 0,C 180,E1 -15367.718,E2 -15367.718} C_VEL
LIN {X 0,Y 326.504,Z 249.279,A -85,B 0,C 180,E1 -15368.702,E2 -15368.702} C_VEL
LIN {X 0,Y 324.949,Z 260.345,A -85,B 0,C 180,E1 -15370.085,E2 -15370.085} C_VEL
LIN {X 0,Y 323.535,Z 270.191,A -85,B 0,C 180,E1 -15371.641,E2 -15371.641} C_VEL
LIN {X 0,Y 322.191,Z 278.251,A -85,B 0,C 180,E1 -15373.201,E2 -15373.201} C_VEL
LIN {X 0,Y 321.041,Z 284.929,A -85,B 0,C 180,E1 -15374.77,E2 -15374.77} C_VEL
LIN {X 0,Y 320.143,Z 291.484,A -85,B 0,C 180,E1 -15376.673,E2 -15376.673} C_VEL
LIN {X 0,Y 319.166,Z 296.703,A -85,B 0,C 180,E1 -15378.57,E2 -15378.57} C_VEL
LIN {X 0,Y 318.624,Z 300.75,A -85,B 0,C 180,E1 -15380.478,E2 -15380.478} C_VEL
LIN {X 0,Y 318.215,Z 303.748,A -85,B 0,C 180,E1 -15382.385,E2 -15382.385} C_VEL
LIN {X 0,Y 317.945,Z 305.618,A -85,B 0,C 180,E1 -15384.104,E2 -15384.104} C_VEL
LIN {X 0,Y 317.894,Z 306.9,A -85,B 0,C 180,E1 -15386.197,E2 -15386.197} C_VEL
LIN {X 0,Y 317.797,Z 307.17,A -85,B 0,C 180,E1 -15387.464,E2 -15387.464} C_VEL
LIN {X 0,Y 317.772,Z 307.047,A -85,B 0,C 180,E1 -15388.732,E2 -15388.732} C_VEL
LIN {X 0,Y 317.857,Z 305.568,A -85,B 0,C 180,E1 -15391.266,E2 -15391.266} C_VEL
LIN {X 0,Y 318.003,Z 304.248,A -85,B 0,C 180,E1 -15392.532,E2 -15392.532} C_VEL
LIN {X 0,Y 318.334,Z 301.458,A -85,B 0,C 180,E1 -15394.431,E2 -15394.431} C_VEL
LIN {X 0,Y 318.789,Z 297.657,A -85,B 0,C 180,E1 -15396.327,E2 -15396.327} C_VEL
LIN {X 0,Y 319.388,Z 292.743,A -85,B 0,C 180,E1 -15398.221,E2 -15398.221} C_VEL
LIN {X 0,Y 320.144,Z 286.563,A -85,B 0,C 180,E1 -15400.113,E2 -15400.113} C_VEL
LIN {X 0,Y 321.331,Z 278.832,A -85,B 0,C 180,E1 -15401.99,E2 -15401.99} C_VEL
LIN {X 0,Y 322.707,Z 269.167,A -85,B 0,C 180,E1 -15403.859,E2 -15403.859} C_VEL
LIN {X 0,Y 323.975,Z 259.161,A -85,B 0,C 180,E1 -15405.409,E2 -15405.409} C_VEL
LIN {X 0,Y 324.942,Z 250.608,A -85,B 0,C 180,E1 -15406.489,E2 -15406.489} C_VEL
LIN {X 0,Y 325.943,Z 241.789,A -85,B 0,C 180,E1 -15407.406,E2 -15407.406} C_VEL
LIN {X 0,Y 326.172,Z 237.17,A -85,B 0,C 180,E1 -15407.835,E2 -15407.835} C_VEL
LIN {X 0,Y 324.391,Z 225.843,A -85,B 0,C 180,E1 -15408.866,E2 -15408.866} C_VEL
LIN {X 0,Y 321.495,Z 213.322,A -85,B 0,C 180,E1 -15409.808,E2 -15409.808} C_VEL
LIN {X 0,Y 318.629,Z 202.819,A -85,B 0,C 180,E1 -15410.469,E2 -15410.469} C_VEL
LIN {X 0,Y 318.813,Z 199.614,A -85,B 0,C 180,E1 -15413.375,E2 -15413.375} C_VEL
LIN {X 0,Y 319.013,Z 196.592,A -85,B 0,C 180,E1 -15416.14,E2 -15416.14} C_VEL
LIN {X 0,Y 319.214,Z 193.6,A -85,B 0,C 180,E1 -15418.968,E2 -15418.968} C_VEL
LIN {X 0,Y 319.424,Z 190.619,A -85,B 0,C 180,E1 -15421.87,E2 -15421.87} C_VEL
LIN {X 0,Y 319.47,Z 187.692,A -85,B 0,C 180,E1 -15424.884,E2 -15424.884} C_VEL
LIN {X 0,Y 319.529,Z 187.683,A -85,B 0,C 180,E1 -15428.01,E2 -15428.01} C_VEL
LIN {X 0,Y 319.515,Z 187.686,A -85,B 0,C 180,E1 -15431.594,E2 -15431.594} C_VEL
LIN {X 0,Y 319.557,Z 187.681,A -85,B 0,C 180,E1 -15435.269,E2 -15435.269} C_VEL
LIN {X 0,Y 319.564,Z 187.678,A -85,B 0,C 180,E1 -15438.717,E2 -15438.717} C_VEL
LIN {X 0,Y 319.564,Z 187.677,A -85,B 0,C 180,E1 -15442.341,E2 -15442.341} C_VEL
LIN {X 0,Y 319.541,Z 187.682,A -85,B 0,C 180,E1 -15445.12,E2 -15445.12} C_VEL
LIN {X 0,Y 319.55,Z 187.681,A -85,B 0,C 180,E1 -15449.056,E2 -15449.056} C_VEL
LIN {X 0,Y 319.587,Z 187.677,A -85,B 0,C 180,E1 -15452.496,E2 -15452.496} C_VEL
LIN {X 0,Y 319.568,Z 187.671,A -85,B 0,C 180,E1 -15455.864,E2 -15455.864} C_VEL
LIN {X 0,Y 318.903,Z 187.755,A -85,B 0,C 180,E1 -15456.915,E2 -15456.915} C_VEL
LIN {X 0,Y 316.069,Z 188.106,A -85,B 0,C 180,E1 -15458.627,E2 -15458.627} C_VEL
LIN {X 0,Y 313.683,Z 188.402,A -85,B 0,C 180,E1 -15460.015,E2 -15460.015} C_VEL
LIN {X 0,Y 312.679,Z 188.529,A -85,B 0,C 180,E1 -15461.089,E2 -15461.089} C_VEL
LIN {X 0,Y 312.607,Z 188.537,A -85,B 0,C 180,E1 -15461.453,E2 -15461.453} C_VEL
LIN {X 0,Y 312.668,Z 188.536,A -85,B 0,C 180,E1 -15465.685,E2 -15465.685} C_VEL
LIN {X 0,Y 312.694,Z 188.53,A -85,B 0,C 180,E1 -15469.641,E2 -15469.641} C_VEL
LIN {X 0,Y 312.862,Z 188.514,A -85,B 0,C 180,E1 -15472.254,E2 -15472.254} C_VEL
LIN {X 0,Y 312.695,Z 188.53,A -85,B 0,C 180,E1 -15474.842,E2 -15474.842} C_VEL
LIN {X 0,Y 312.96,Z 188.498,A -85,B 0,C 180,E1 -15478.713,E2 -15478.713} C_VEL
LIN {X 0,Y 312.965,Z 188.5,A -85,B 0,C 180,E1 -15481.286,E2 -15481.286} C_VEL
LIN {X 0,Y 312.687,Z 188.536,A -85,B 0,C 180,E1 -15483.866,E2 -15483.866} C_VEL
LIN {X 0,Y 312.884,Z 188.508,A -85,B 0,C 180,E1 -15486.448,E2 -15486.448} C_VEL
LIN {X 0,Y 312.761,Z 188.526,A -85,B 0,C 180,E1 -15489.05,E2 -15489.05} C_VEL
LIN {X 0,Y 312.608,Z 188.545,A -85,B 0,C 180,E1 -15492.992,E2 -15492.992} C_VEL
LIN {X 0,Y 312.6,Z 188.546,A -85,B 0,C 180,E1 -15495.651,E2 -15495.651} C_VEL
LIN {X 0,Y 312.587,Z 188.547,A -85,B 0,C 180,E1 -15499.709,E2 -15499.709} C_VEL
LIN {X 0,Y 312.549,Z 188.554,A -85,B 0,C 180,E1 -15502.802,E2 -15502.802} C_VEL
LIN {X 0,Y 312.532,Z 188.556,A -85,B 0,C 180,E1 -15506.727,E2 -15506.727} C_VEL
LIN {X 0,Y 312.523,Z 188.551,A -85,B 0,C 180,E1 -15509.652,E2 -15509.652} C_VEL
LIN {X 0,Y 312.499,Z 188.556,A -85,B 0,C 180,E1 -15513.691,E2 -15513.691} C_VEL
LIN {X 0,Y 312.521,Z 188.554,A -85,B 0,C 180,E1 -15517.386,E2 -15517.386} C_VEL
LIN {X 0,Y 312.51,Z 188.559,A -85,B 0,C 180,E1 -15520.706,E2 -15520.706} C_VEL
LIN {X 0,Y 312.58,Z 188.551,A -85,B 0,C 180,E1 -15524.187,E2 -15524.187} C_VEL
LIN {X 0,Y 312.619,Z 188.618,A -85,B 0,C 180,E1 -15525.427,E2 -15525.427} C_VEL
LIN {X 0,Y 313.075,Z 191.394,A -85,B 0,C 180,E1 -15527.799,E2 -15527.799} C_VEL
LIN {X 0,Y 313.78,Z 196.105,A -85,B 0,C 180,E1 -15531.621,E2 -15531.621} C_VEL
LIN {X 0,Y 313.944,Z 199.78,A -85,B 0,C 180,E1 -15534.41,E2 -15534.41} C_VEL
LIN {X 0,Y 313.476,Z 204.018,A -85,B 0,C 180,E1 -15537.451,E2 -15537.451} C_VEL
LIN {X 0,Y 312.769,Z 209.413,A -85,B 0,C 180,E1 -15541.204,E2 -15541.204} C_VEL
LIN {X 0,Y 312.07,Z 215.569,A -85,B 0,C 180,E1 -15545.381,E2 -15545.381} C_VEL
LIN {X 0,Y 311.848,Z 218.093,A -85,B 0,C 180,E1 -15547.069,E2 -15547.069} C_VEL
LIN {X 0,Y 314.831,Z 231.93,A -85,B 0,C 180,E1 -15547.88,E2 -15547.88} C_VEL
LIN {X 0,Y 316.7,Z 243.709,A -85,B 0,C 180,E1 -15548.754,E2 -15548.754} C_VEL
LIN {X 0,Y 317.936,Z 255.147,A -85,B 0,C 180,E1 -15549.797,E2 -15549.797} C_VEL
LIN {X 0,Y 318.127,Z 261.776,A -85,B 0,C 180,E1 -15550.482,E2 -15550.482} C_VEL
LIN {X 0,Y 316.743,Z 272.631,A -85,B 0,C 180,E1 -15551.737,E2 -15551.737} C_VEL
LIN {X 0,Y 315.399,Z 282.48,A -85,B 0,C 180,E1 -15553.164,E2 -15553.164} C_VEL
LIN {X 0,Y 314.216,Z 291.444,A -85,B 0,C 180,E1 -15554.765,E2 -15554.765} C_VEL
LIN {X 0,Y 313.012,Z 300.197,A -85,B 0,C 180,E1 -15556.697,E2 -15556.697} C_VEL
LIN {X 0,Y 312.001,Z 307.173,A -85,B 0,C 180,E1 -15558.634,E2 -15558.634} C_VEL
LIN {X 0,Y 311.289,Z 313.58,A -85,B 0,C 180,E1 -15560.908,E2 -15560.908} C_VEL
LIN {X 0,Y 310.933,Z 317.787,A -85,B 0,C 180,E1 -15562.86,E2 -15562.86} C_VEL
LIN {X 0,Y 310.713,Z 320.928,A -85,B 0,C 180,E1 -15564.81,E2 -15564.81} C_VEL
LIN {X 0,Y 310.719,Z 322.496,A -85,B 0,C 180,E1 -15566.11,E2 -15566.11} C_VEL
LIN {X 0,Y 310.682,Z 323.623,A -85,B 0,C 180,E1 -15567.408,E2 -15567.408} C_VEL
LIN {X 0,Y 310.69,Z 324.652,A -85,B 0,C 180,E1 -15570.001,E2 -15570.001} C_VEL
LIN {X 0,Y 310.648,Z 324.585,A -85,B 0,C 180,E1 -15571.297,E2 -15571.297} C_VEL
LIN {X 0,Y 310.677,Z 324.111,A -85,B 0,C 180,E1 -15572.594,E2 -15572.594} C_VEL
LIN {X 0,Y 310.696,Z 323.211,A -85,B 0,C 180,E1 -15573.892,E2 -15573.892} C_VEL
LIN {X 0,Y 310.821,Z 320.222,A -85,B 0,C 180,E1 -15576.492,E2 -15576.492} C_VEL
LIN {X 0,Y 311.191,Z 316.817,A -85,B 0,C 180,E1 -15578.442,E2 -15578.442} C_VEL
LIN {X 0,Y 311.738,Z 312.34,A -85,B 0,C 180,E1 -15580.391,E2 -15580.391} C_VEL
LIN {X 0,Y 312.712,Z 305.572,A -85,B 0,C 180,E1 -15582.658,E2 -15582.658} C_VEL
LIN {X 0,Y 314.063,Z 298.214,A -85,B 0,C 180,E1 -15584.581,E2 -15584.581} C_VEL
LIN {X 0,Y 315.412,Z 289.324,A -85,B 0,C 180,E1 -15586.458,E2 -15586.458} C_VEL
LIN {X 0,Y 316.909,Z 279.617,A -85,B 0,C 180,E1 -15588.087,E2 -15588.087} C_VEL
LIN {X 0,Y 318.527,Z 269.119,A -85,B 0,C 180,E1 -15589.494,E2 -15589.494} C_VEL
LIN {X 0,Y 319.49,Z 262.183,A -85,B 0,C 180,E1 -15590.27,E2 -15590.27} C_VEL
LIN {X 0,Y 318.707,Z 251.68,A -85,B 0,C 180,E1 -15591.379,E2 -15591.379} C_VEL
LIN {X 0,Y 316.874,Z 239.076,A -85,B 0,C 180,E1 -15592.493,E2 -15592.493} C_VEL
LIN {X 0,Y 314.088,Z 225.867,A -85,B 0,C 180,E1 -15593.449,E2 -15593.449} C_VEL
LIN {X 0,Y 312.107,Z 217.91,A -85,B 0,C 180,E1 -15593.955,E2 -15593.955} C_VEL
LIN {X 0,Y 312.791,Z 211.77,A -85,B 0,C 180,E1 -15598.153,E2 -15598.153} C_VEL
LIN {X 0,Y 313.499,Z 206.9,A -85,B 0,C 180,E1 -15601.583,E2 -15601.583} C_VEL
LIN {X 0,Y 313.996,Z 203.419,A -85,B 0,C 180,E1 -15604.091,E2 -15604.091} C_VEL
LIN {X 0,Y 314.142,Z 199.345,A -85,B 0,C 180,E1 -15607.158,E2 -15607.158} C_VEL
LIN {X 0,Y 313.687,Z 195.167,A -85,B 0,C 180,E1 -15610.519,E2 -15610.519} C_VEL
LIN {X 0,Y 313.02,Z 191.007,A -85,B 0,C 180,E1 -15614.106,E2 -15614.106} C_VEL
LIN {X 0,Y 312.525,Z 188.561,A -85,B 0,C 180,E1 -15616.4,E2 -15616.4} C_VEL
LIN {X 0,Y 312.494,Z 188.56,A -85,B 0,C 180,E1 -15619.873,E2 -15619.873} C_VEL
LIN {X 0,Y 312.522,Z 188.556,A -85,B 0,C 180,E1 -15624.05,E2 -15624.05} C_VEL
LIN {X 0,Y 312.488,Z 188.564,A -85,B 0,C 180,E1 -15627.332,E2 -15627.332} C_VEL
LIN {X 0,Y 312.553,Z 188.551,A -85,B 0,C 180,E1 -15631.823,E2 -15631.823} C_VEL
LIN {X 0,Y 312.572,Z 188.55,A -85,B 0,C 180,E1 -15634.71,E2 -15634.71} C_VEL
LIN {X 0,Y 312.589,Z 188.546,A -85,B 0,C 180,E1 -15637.529,E2 -15637.529} C_VEL
LIN {X 0,Y 312.622,Z 188.541,A -85,B 0,C 180,E1 -15641.656,E2 -15641.656} C_VEL
LIN {X 0,Y 312.675,Z 188.534,A -85,B 0,C 180,E1 -15645.686,E2 -15645.686} C_VEL
LIN {X 0,Y 312.684,Z 188.533,A -85,B 0,C 180,E1 -15649.641,E2 -15649.641} C_VEL
LIN {X 0,Y 312.839,Z 188.517,A -85,B 0,C 180,E1 -15652.254,E2 -15652.254} C_VEL
LIN {X 0,Y 312.701,Z 188.532,A -85,B 0,C 180,E1 -15654.842,E2 -15654.842} C_VEL
LIN {X 0,Y 312.966,Z 188.5,A -85,B 0,C 180,E1 -15658.714,E2 -15658.714} C_VEL
LIN {X 0,Y 312.974,Z 188.497,A -85,B 0,C 180,E1 -15661.287,E2 -15661.287} C_VEL
LIN {X 0,Y 312.695,Z 188.535,A -85,B 0,C 180,E1 -15663.867,E2 -15663.867} C_VEL
LIN {X 0,Y 312.873,Z 188.511,A -85,B 0,C 180,E1 -15666.55,E2 -15666.55} C_VEL
LIN {X 0,Y 312.735,Z 188.526,A -85,B 0,C 180,E1 -15669.051,E2 -15669.051} C_VEL
LIN {X 0,Y 312.614,Z 188.542,A -85,B 0,C 180,E1 -15672.992,E2 -15672.992} C_VEL
LIN {X 0,Y 312.623,Z 188.545,A -85,B 0,C 180,E1 -15675.651,E2 -15675.651} C_VEL
LIN {X 0,Y 312.615,Z 188.544,A -85,B 0,C 180,E1 -15679.237,E2 -15679.237} C_VEL
LIN {X 0,Y 312.531,Z 188.553,A -85,B 0,C 180,E1 -15682.79,E2 -15682.79} C_VEL
LIN {X 0,Y 312.583,Z 188.546,A -85,B 0,C 180,E1 -15685.935,E2 -15685.935} C_VEL
LIN {X 0,Y 312.532,Z 188.554,A -85,B 0,C 180,E1 -15689.652,E2 -15689.652} C_VEL
LIN {X 0,Y 312.509,Z 188.556,A -85,B 0,C 180,E1 -15693.69,E2 -15693.69} C_VEL
LIN {X 0,Y 312.509,Z 188.557,A -85,B 0,C 180,E1 -15697.388,E2 -15697.388} C_VEL
LIN {X 0,Y 312.481,Z 188.562,A -85,B 0,C 180,E1 -15700.711,E2 -15700.711} C_VEL
LIN {X 0,Y 312.444,Z 188.565,A -85,B 0,C 180,E1 -15704.212,E2 -15704.212} C_VEL
LIN {X 0,Y 312.449,Z 188.565,A -85,B 0,C 180,E1 -15707.927,E2 -15707.927} C_VEL
LIN {X 0,Y 312.421,Z 188.57,A -85,B 0,C 180,E1 -15709.282,E2 -15709.282} C_VEL
LIN {X 0,Y 312.656,Z 191.478,A -85,B 0,C 180,E1 -15712.635,E2 -15712.635} C_VEL
LIN {X 0,Y 312.454,Z 194.533,A -85,B 0,C 180,E1 -15715.785,E2 -15715.785} C_VEL
LIN {X 0,Y 312.172,Z 197.571,A -85,B 0,C 180,E1 -15718.816,E2 -15718.816} C_VEL
LIN {X 0,Y 311.947,Z 200.645,A -85,B 0,C 180,E1 -15721.764,E2 -15721.764} C_VEL
LIN {X 0,Y 311.786,Z 203.275,A -85,B 0,C 180,E1 -15724.135,E2 -15724.135} C_VEL
LIN {X 0,Y 315.778,Z 216.444,A -85,B 0,C 180,E1 -15725.066,E2 -15725.066} C_VEL
LIN {X 0,Y 318.766,Z 228.999,A -85,B 0,C 180,E1 -15726.146,E2 -15726.146} C_VEL
LIN {X 0,Y 320.701,Z 240.095,A -85,B 0,C 180,E1 -15727.279,E2 -15727.279} C_VEL
LIN {X 0,Y 320.29,Z 246.395,A -85,B 0,C 180,E1 -15727.928,E2 -15727.928} C_VEL
LIN {X 0,Y 318.8,Z 256.93,A -85,B 0,C 180,E1 -15729.178,E2 -15729.178} C_VEL
LIN {X 0,Y 317.31,Z 266.546,A -85,B 0,C 180,E1 -15730.596,E2 -15730.596} C_VEL
LIN {X 0,Y 315.847,Z 275.3,A -85,B 0,C 180,E1 -15732.185,E2 -15732.185} C_VEL
LIN {X 0,Y 314.45,Z 283.241,A -85,B 0,C 180,E1 -15733.959,E2 -15733.959} C_VEL
LIN {X 0,Y 313.364,Z 290.601,A -85,B 0,C 180,E1 -15736.049,E2 -15736.049} C_VEL
LIN {X 0,Y 312.164,Z 296.839,A -85,B 0,C 180,E1 -15738.31,E2 -15738.31} C_VEL
LIN {X 0,Y 311.606,Z 300.9,A -85,B 0,C 180,E1 -15740.261,E2 -15740.261} C_VEL
LIN {X 0,Y 311.176,Z 303.911,A -85,B 0,C 180,E1 -15742.211,E2 -15742.211} C_VEL
LIN {X 0,Y 310.861,Z 305.937,A -85,B 0,C 180,E1 -15744.137,E2 -15744.137} C_VEL
LIN {X 0,Y 310.803,Z 307.089,A -85,B 0,C 180,E1 -15746.11,E2 -15746.11} C_VEL
LIN {X 0,Y 310.721,Z 307.364,A -85,B 0,C 180,E1 -15747.407,E2 -15747.407} C_VEL
LIN {X 0,Y 310.685,Z 307.252,A -85,B 0,C 180,E1 -15748.703,E2 -15748.703} C_VEL
LIN {X 0,Y 310.769,Z 305.787,A -85,B 0,C 180,E1 -15751.295,E2 -15751.295} C_VEL
LIN {X 0,Y 310.922,Z 304.474,A -85,B 0,C 180,E1 -15752.59,E2 -15752.59} C_VEL
LIN {X 0,Y 311.274,Z 301.696,A -85,B 0,C 180,E1 -15754.531,E2 -15754.531} C_VEL
LIN {X 0,Y 311.748,Z 297.91,A -85,B 0,C 180,E1 -15756.471,E2 -15756.471} C_VEL
LIN {X 0,Y 312.383,Z 293.01,A -85,B 0,C 180,E1 -15758.407,E2 -15758.407} C_VEL
LIN {X 0,Y 313.167,Z 286.847,A -85,B 0,C 180,E1 -15760.341,E2 -15760.341} C_VEL
LIN {X 0,Y 314.403,Z 279.144,A -85,B 0,C 180,E1 -15762.259,E2 -15762.259} C_VEL
LIN {X 0,Y 315.82,Z 269.502,A -85,B 0,C 180,E1 -15764.167,E2 -15764.167} C_VEL
LIN {X 0,Y 317.158,Z 259.533,A -85,B 0,C 180,E1 -15765.749,E2 -15765.749} C_VEL
LIN {X 0,Y 318.178,Z 251.003,A -85,B 0,C 180,E1 -15766.85,E2 -15766.85} C_VEL
LIN {X 0,Y 319.196,Z 242.229,A -85,B 0,C 180,E1 -15767.786,E2 -15767.786} C_VEL
LIN {X 0,Y 319.291,Z 237.65,A -85,B 0,C 180,E1 -15768.233,E2 -15768.233} C_VEL
LIN {X 0,Y 317.567,Z 226.873,A -85,B 0,C 180,E1 -15769.252,E2 -15769.252} C_VEL
LIN {X 0,Y 314.776,Z 214.517,A -85,B 0,C 180,E1 -15770.227,E2 -15770.227} C_VEL
LIN {X 0,Y 311.588,Z 203.017,A -85,B 0,C 180,E1 -15770.992,E2 -15770.992} C_VEL
LIN {X 0,Y 311.797,Z 199.816,A -85,B 0,C 180,E1 -15773.934,E2 -15773.934} C_VEL
LIN {X 0,Y 311.996,Z 196.823,A -85,B 0,C 180,E1 -15776.774,E2 -15776.774} C_VEL
LIN {X 0,Y 312.227,Z 193.8,A -85,B 0,C 180,E1 -15779.68,E2 -15779.68} C_VEL
LIN {X 0,Y 312.416,Z 190.817,A -85,B 0,C 180,E1 -15782.673,E2 -15782.673} C_VEL
LIN {X 0,Y 312.431,Z 189.347,A -85,B 0,C 180,E1 -15784.216,E2 -15784.216} C_VEL
LIN {X 0,Y 312.497,Z 188.561,A -85,B 0,C 180,E1 -15785.939,E2 -15785.939} C_VEL
LIN {X 0,Y 312.494,Z 188.558,A -85,B 0,C 180,E1 -15790.122,E2 -15790.122} C_VEL
LIN {X 0,Y 312.506,Z 188.556,A -85,B 0,C 180,E1 -15794.195,E2 -15794.195} C_VEL
LIN {X 0,Y 312.533,Z 188.553,A -85,B 0,C 180,E1 -15797.903,E2 -15797.903} C_VEL
LIN {X 0,Y 312.526,Z 188.553,A -85,B 0,C 180,E1 -15801.906,E2 -15801.906} C_VEL
LIN {X 0,Y 312.487,Z 188.558,A -85,B 0,C 180,E1 -15805.787,E2 -15805.787} C_VEL
LIN {X 0,Y 312.503,Z 188.56,A -85,B 0,C 180,E1 -15808.851,E2 -15808.851} C_VEL
LIN {X 0,Y 312.553,Z 188.549,A -85,B 0,C 180,E1 -15811.822,E2 -15811.822} C_VEL
LIN {X 0,Y 312.566,Z 188.55,A -85,B 0,C 180,E1 -15814.709,E2 -15814.709} C_VEL
LIN {X 0,Y 312.582,Z 188.539,A -85,B 0,C 180,E1 -15817.528,E2 -15817.528} C_VEL
LIN {X 0,Y 312.607,Z 188.537,A -85,B 0,C 180,E1 -15821.453,E2 -15821.453} C_VEL
LIN {X 0,Y 311.965,Z 188.624,A -85,B 0,C 180,E1 -15822.529,E2 -15822.529} C_VEL
LIN {X 0,Y 309.115,Z 188.981,A -85,B 0,C 180,E1 -15824.281,E2 -15824.281} C_VEL
LIN {X 0,Y 306.682,Z 189.283,A -85,B 0,C 180,E1 -15825.702,E2 -15825.702} C_VEL
LIN {X 0,Y 305.638,Z 189.411,A -85,B 0,C 180,E1 -15826.803,E2 -15826.803} C_VEL
LIN {X 0,Y 305.554,Z 189.42,A -85,B 0,C 180,E1 -15827.176,E2 -15827.176} C_VEL
LIN {X 0,Y 305.791,Z 189.391,A -85,B 0,C 180,E1 -15831.183,E2 -15831.183} C_VEL
LIN {X 0,Y 305.834,Z 189.387,A -85,B 0,C 180,E1 -15833.402,E2 -15833.402} C_VEL
LIN {X 0,Y 305.927,Z 189.375,A -85,B 0,C 180,E1 -15838.683,E2 -15838.683} C_VEL
LIN {X 0,Y 305.932,Z 189.376,A -85,B 0,C 180,E1 -15841.316,E2 -15841.316} C_VEL
LIN {X 0,Y 305.668,Z 189.41,A -85,B 0,C 180,E1 -15845.277,E2 -15845.277} C_VEL
LIN {X 0,Y 305.786,Z 189.395,A -85,B 0,C 180,E1 -15847.926,E2 -15847.926} C_VEL
LIN {X 0,Y 305.579,Z 189.42,A -85,B 0,C 180,E1 -15851.946,E2 -15851.946} C_VEL
LIN {X 0,Y 305.594,Z 189.419,A -85,B 0,C 180,E1 -15855.023,E2 -15855.023} C_VEL
LIN {X 0,Y 305.579,Z 189.421,A -85,B 0,C 180,E1 -15859.46,E2 -15859.46} C_VEL
LIN {X 0,Y 305.501,Z 189.433,A -85,B 0,C 180,E1 -15863.058,E2 -15863.058} C_VEL
LIN {X 0,Y 305.525,Z 189.426,A -85,B 0,C 180,E1 -15866.229,E2 -15866.229} C_VEL
LIN {X 0,Y 305.473,Z 189.432,A -85,B 0,C 180,E1 -15869.051,E2 -15869.051} C_VEL
LIN {X 0,Y 305.444,Z 189.435,A -85,B 0,C 180,E1 -15873.519,E2 -15873.519} C_VEL
LIN {X 0,Y 305.478,Z 189.435,A -85,B 0,C 180,E1 -15876.739,E2 -15876.739} C_VEL
LIN {X 0,Y 305.469,Z 189.436,A -85,B 0,C 180,E1 -15880.609,E2 -15880.609} C_VEL
LIN {X 0,Y 305.54,Z 189.427,A -85,B 0,C 180,E1 -15884.521,E2 -15884.521} C_VEL
LIN {X 0,Y 305.598,Z 189.657,A -85,B 0,C 180,E1 -15885.203,E2 -15885.203} C_VEL
LIN {X 0,Y 306.338,Z 194.28,A -85,B 0,C 180,E1 -15889.208,E2 -15889.208} C_VEL
LIN {X 0,Y 306.803,Z 197.444,A -85,B 0,C 180,E1 -15891.798,E2 -15891.798} C_VEL
LIN {X 0,Y 306.926,Z 200.631,A -85,B 0,C 180,E1 -15894.279,E2 -15894.279} C_VEL
LIN {X 0,Y 306.45,Z 204.862,A -85,B 0,C 180,E1 -15897.393,E2 -15897.393} C_VEL
LIN {X 0,Y 305.725,Z 210.125,A -85,B 0,C 180,E1 -15901.138,E2 -15901.138} C_VEL
LIN {X 0,Y 304.988,Z 216.381,A -85,B 0,C 180,E1 -15905.497,E2 -15905.497} C_VEL
LIN {X 0,Y 304.855,Z 217.867,A -85,B 0,C 180,E1 -15906.523,E2 -15906.523} C_VEL
LIN {X 0,Y 308.074,Z 232.742,A -85,B 0,C 180,E1 -15907.449,E2 -15907.449} C_VEL
LIN {X 0,Y 309.939,Z 244.785,A -85,B 0,C 180,E1 -15908.387,E2 -15908.387} C_VEL
LIN {X 0,Y 311.168,Z 256.682,A -85,B 0,C 180,E1 -15909.527,E2 -15909.527} C_VEL
LIN {X 0,Y 311.233,Z 262.889,A -85,B 0,C 180,E1 -15910.204,E2 -15910.204} C_VEL
LIN {X 0,Y 309.654,Z 274.647,A -85,B 0,C 180,E1 -15911.647,E2 -15911.647} C_VEL
LIN {X 0,Y 308.355,Z 283.812,A -85,B 0,C 180,E1 -15913.054,E2 -15913.054} C_VEL
LIN {X 0,Y 307.09,Z 292.775,A -85,B 0,C 180,E1 -15914.743,E2 -15914.743} C_VEL
LIN {X 0,Y 305.853,Z 301.167,A -85,B 0,C 180,E1 -15916.718,E2 -15916.718} C_VEL
LIN {X 0,Y 304.882,Z 307.928,A -85,B 0,C 180,E1 -15918.702,E2 -15918.702} C_VEL
LIN {X 0,Y 304.244,Z 313.332,A -85,B 0,C 180,E1 -15920.696,E2 -15920.696} C_VEL
LIN {X 0,Y 303.852,Z 317.551,A -85,B 0,C 180,E1 -15922.693,E2 -15922.693} C_VEL
LIN {X 0,Y 303.636,Z 320.703,A -85,B 0,C 180,E1 -15924.689,E2 -15924.689} C_VEL
LIN {X 0,Y 303.632,Z 322.276,A -85,B 0,C 180,E1 -15926.019,E2 -15926.019} C_VEL
LIN {X 0,Y 303.607,Z 323.414,A -85,B 0,C 180,E1 -15927.348,E2 -15927.348} C_VEL
LIN {X 0,Y 303.603,Z 324.452,A -85,B 0,C 180,E1 -15930.001,E2 -15930.001} C_VEL
LIN {X 0,Y 303.565,Z 324.39,A -85,B 0,C 180,E1 -15931.327,E2 -15931.327} C_VEL
LIN {X 0,Y 303.602,Z 323.925,A -85,B 0,C 180,E1 -15932.654,E2 -15932.654} C_VEL
LIN {X 0,Y 303.592,Z 323.03,A -85,B 0,C 180,E1 -15933.983,E2 -15933.983} C_VEL
LIN {X 0,Y 303.617,Z 321.502,A -85,B 0,C 180,E1 -15935.53,E2 -15935.53} C_VEL
LIN {X 0,Y 303.99,Z 317.907,A -85,B 0,C 180,E1 -15937.974,E2 -15937.974} C_VEL
LIN {X 0,Y 304.492,Z 313.812,A -85,B 0,C 180,E1 -15939.969,E2 -15939.969} C_VEL
LIN {X 0,Y 305.434,Z 307.544,A -85,B 0,C 180,E1 -15942.289,E2 -15942.289} C_VEL
LIN {X 0,Y 306.671,Z 300.733,A -85,B 0,C 180,E1 -15944.262,E2 -15944.262} C_VEL
LIN {X 0,Y 308.012,Z 292.716,A -85,B 0,C 180,E1 -15946.134,E2 -15946.134} C_VEL
LIN {X 0,Y 309.486,Z 283.546,A -85,B 0,C 180,E1 -15947.852,E2 -15947.852} C_VEL
LIN {X 0,Y 311.226,Z 272.832,A -85,B 0,C 180,E1 -15949.455,E2 -15949.455} C_VEL
LIN {X 0,Y 312.733,Z 262.168,A -85,B 0,C 180,E1 -15950.728,E2 -15950.728} C_VEL
LIN {X 0,Y 311.655,Z 249.969,A -85,B 0,C 180,E1 -15952.042,E2 -15952.042} C_VEL
LIN {X 0,Y 309.852,Z 238.294,A -85,B 0,C 180,E1 -15953.094,E2 -15953.094} C_VEL
LIN {X 0,Y 307.157,Z 225.726,A -85,B 0,C 180,E1 -15954.031,E2 -15954.031} C_VEL
LIN {X 0,Y 305.127,Z 217.738,A -85,B 0,C 180,E1 -15954.538,E2 -15954.538} C_VEL
LIN {X 0,Y 305.969,Z 211.118,A -85,B 0,C 180,E1 -15959.209,E2 -15959.209} C_VEL
LIN {X 0,Y 306.508,Z 207.303,A -85,B 0,C 180,E1 -15961.964,E2 -15961.964} C_VEL
LIN {X 0,Y 307.017,Z 203.365,A -85,B 0,C 180,E1 -15964.908,E2 -15964.908} C_VEL
LIN {X 0,Y 307.12,Z 200.943,A -85,B 0,C 180,E1 -15966.782,E2 -15966.782} C_VEL
LIN {X 0,Y 306.766,Z 197.14,A -85,B 0,C 180,E1 -15969.9,E2 -15969.9} C_VEL
LIN {X 0,Y 306.15,Z 192.948,A -85,B 0,C 180,E1 -15973.523,E2 -15973.523} C_VEL
LIN {X 0,Y 305.473,Z 189.438,A -85,B 0,C 180,E1 -15976.942,E2 -15976.942} C_VEL
LIN {X 0,Y 305.448,Z 189.438,A -85,B 0,C 180,E1 -15979.891,E2 -15979.891} C_VEL
LIN {X 0,Y 305.469,Z 189.437,A -85,B 0,C 180,E1 -15983.631,E2 -15983.631} C_VEL
LIN {X 0,Y 305.452,Z 189.436,A -85,B 0,C 180,E1 -15986.482,E2 -15986.482} C_VEL
LIN {X 0,Y 305.465,Z 189.437,A -85,B 0,C 180,E1 -15990.955,E2 -15990.955} C_VEL
LIN {X 0,Y 305.55,Z 189.422,A -85,B 0,C 180,E1 -15994.086,E2 -15994.086} C_VEL
LIN {X 0,Y 305.527,Z 189.427,A -85,B 0,C 180,E1 -15998.405,E2 -15998.405} C_VEL
LIN {X 0,Y 305.577,Z 189.421,A -85,B 0,C 180,E1 -16001.217,E2 -16001.217} C_VEL
LIN {X 0,Y 305.631,Z 189.412,A -85,B 0,C 180,E1 -16005.348,E2 -16005.348} C_VEL
LIN {X 0,Y 305.621,Z 189.413,A -85,B 0,C 180,E1 -16009.399,E2 -16009.399} C_VEL
LIN {X 0,Y 305.782,Z 189.395,A -85,B 0,C 180,E1 -16012.074,E2 -16012.074} C_VEL
LIN {X 0,Y 305.672,Z 189.409,A -85,B 0,C 180,E1 -16014.723,E2 -16014.723} C_VEL
LIN {X 0,Y 305.934,Z 189.376,A -85,B 0,C 180,E1 -16018.684,E2 -16018.684} C_VEL
LIN {X 0,Y 305.942,Z 189.373,A -85,B 0,C 180,E1 -16021.317,E2 -16021.317} C_VEL
LIN {X 0,Y 305.674,Z 189.407,A -85,B 0,C 180,E1 -16025.277,E2 -16025.277} C_VEL
LIN {X 0,Y 305.77,Z 189.399,A -85,B 0,C 180,E1 -16027.927,E2 -16027.927} C_VEL
LIN {X 0,Y 305.579,Z 189.422,A -85,B 0,C 180,E1 -16031.946,E2 -16031.946} C_VEL
LIN {X 0,Y 305.622,Z 189.413,A -85,B 0,C 180,E1 -16035.035,E2 -16035.035} C_VEL
LIN {X 0,Y 305.561,Z 189.425,A -85,B 0,C 180,E1 -16039.446,E2 -16039.446} C_VEL
LIN {X 0,Y 305.476,Z 189.433,A -85,B 0,C 180,E1 -16043.042,E2 -16043.042} C_VEL
LIN {X 0,Y 305.512,Z 189.426,A -85,B 0,C 180,E1 -16046.22,E2 -16046.22} C_VEL
LIN {X 0,Y 305.483,Z 189.433,A -85,B 0,C 180,E1 -16049.051,E2 -16049.051} C_VEL
LIN {X 0,Y 305.454,Z 189.436,A -85,B 0,C 180,E1 -16053.519,E2 -16053.519} C_VEL
LIN {X 0,Y 305.462,Z 189.436,A -85,B 0,C 180,E1 -16056.742,E2 -16056.742} C_VEL
LIN {X 0,Y 305.446,Z 189.437,A -85,B 0,C 180,E1 -16060.601,E2 -16060.601} C_VEL
LIN {X 0,Y 305.418,Z 189.439,A -85,B 0,C 180,E1 -16063.657,E2 -16063.657} C_VEL
LIN {X 0,Y 305.429,Z 189.44,A -85,B 0,C 180,E1 -16067.42,E2 -16067.42} C_VEL
LIN {X 0,Y 305.412,Z 189.698,A -85,B 0,C 180,E1 -16069.411,E2 -16069.411} C_VEL
LIN {X 0,Y 305.598,Z 191.628,A -85,B 0,C 180,E1 -16071.618,E2 -16071.618} C_VEL
LIN {X 0,Y 305.499,Z 194.682,A -85,B 0,C 180,E1 -16074.894,E2 -16074.894} C_VEL
LIN {X 0,Y 305.154,Z 198.183,A -85,B 0,C 180,E1 -16078.447,E2 -16078.447} C_VEL
LIN {X 0,Y 304.812,Z 202.322,A -85,B 0,C 180,E1 -16082.541,E2 -16082.541} C_VEL
LIN {X 0,Y 304.754,Z 203.334,A -85,B 0,C 180,E1 -16083.51,E2 -16083.51} C_VEL
LIN {X 0,Y 309.009,Z 217.2,A -85,B 0,C 180,E1 -16084.542,E2 -16084.542} C_VEL
LIN {X 0,Y 312.042,Z 229.823,A -85,B 0,C 180,E1 -16085.675,E2 -16085.675} C_VEL
LIN {X 0,Y 313.885,Z 240.6,A -85,B 0,C 180,E1 -16086.815,E2 -16086.815} C_VEL
LIN {X 0,Y 313.967,Z 243.791,A -85,B 0,C 180,E1 -16087.169,E2 -16087.169} C_VEL
LIN {X 0,Y 312.517,Z 254.531,A -85,B 0,C 180,E1 -16088.393,E2 -16088.393} C_VEL
LIN {X 0,Y 310.89,Z 264.645,A -85,B 0,C 180,E1 -16089.835,E2 -16089.835} C_VEL
LIN {X 0,Y 309.376,Z 273.748,A -85,B 0,C 180,E1 -16091.456,E2 -16091.456} C_VEL
LIN {X 0,Y 307.739,Z 282.556,A -85,B 0,C 180,E1 -16093.4,E2 -16093.4} C_VEL
LIN {X 0,Y 306.642,Z 289.714,A -85,B 0,C 180,E1 -16095.398,E2 -16095.398} C_VEL
LIN {X 0,Y 305.506,Z 295.369,A -85,B 0,C 180,E1 -16097.377,E2 -16097.377} C_VEL
LIN {X 0,Y 304.747,Z 299.816,A -85,B 0,C 180,E1 -16099.368,E2 -16099.368} C_VEL
LIN {X 0,Y 304.405,Z 302.159,A -85,B 0,C 180,E1 -16100.699,E2 -16100.699} C_VEL
LIN {X 0,Y 304.11,Z 304.075,A -85,B 0,C 180,E1 -16102.029,E2 -16102.029} C_VEL
LIN {X 0,Y 303.776,Z 306.259,A -85,B 0,C 180,E1 -16104.174,E2 -16104.174} C_VEL
LIN {X 0,Y 303.715,Z 307.277,A -85,B 0,C 180,E1 -16106.019,E2 -16106.019} C_VEL
LIN {X 0,Y 303.647,Z 307.558,A -85,B 0,C 180,E1 -16107.346,E2 -16107.346} C_VEL
LIN {X 0,Y 303.601,Z 307.455,A -85,B 0,C 180,E1 -16108.673,E2 -16108.673} C_VEL
LIN {X 0,Y 303.613,Z 306.926,A -85,B 0,C 180,E1 -16109.999,E2 -16109.999} C_VEL
LIN {X 0,Y 303.844,Z 304.699,A -85,B 0,C 180,E1 -16112.65,E2 -16112.65} C_VEL
LIN {X 0,Y 304.219,Z 301.934,A -85,B 0,C 180,E1 -16114.637,E2 -16114.637} C_VEL
LIN {X 0,Y 304.707,Z 298.162,A -85,B 0,C 180,E1 -16116.621,E2 -16116.621} C_VEL
LIN {X 0,Y 305.376,Z 293.275,A -85,B 0,C 180,E1 -16118.602,E2 -16118.602} C_VEL
LIN {X 0,Y 306.204,Z 287.13,A -85,B 0,C 180,E1 -16120.579,E2 -16120.579} C_VEL
LIN {X 0,Y 307.473,Z 279.456,A -85,B 0,C 180,E1 -16122.54,E2 -16122.54} C_VEL
LIN {X 0,Y 308.949,Z 269.836,A -85,B 0,C 180,E1 -16124.489,E2 -16124.489} C_VEL
LIN {X 0,Y 310.349,Z 259.901,A -85,B 0,C 180,E1 -16126.103,E2 -16126.103} C_VEL
LIN {X 0,Y 311.412,Z 251.398,A -85,B 0,C 180,E1 -16127.228,E2 -16127.228} C_VEL
LIN {X 0,Y 312.463,Z 242.669,A -85,B 0,C 180,E1 -16128.182,E2 -16128.182} C_VEL
LIN {X 0,Y 312.559,Z 239.199,A -85,B 0,C 180,E1 -16128.535,E2 -16128.535} C_VEL
LIN {X 0,Y 310.805,Z 227.794,A -85,B 0,C 180,E1 -16129.659,E2 -16129.659} C_VEL
LIN {X 0,Y 307.992,Z 215.465,A -85,B 0,C 180,E1 -16130.678,E2 -16130.678} C_VEL
LIN {X 0,Y 304.552,Z 203.246,A -85,B 0,C 180,E1 -16131.486,E2 -16131.486} C_VEL
LIN {X 0,Y 304.798,Z 200.06,A -85,B 0,C 180,E1 -16134.519,E2 -16134.519} C_VEL
LIN {X 0,Y 304.997,Z 197.02,A -85,B 0,C 180,E1 -16137.439,E2 -16137.439} C_VEL
LIN {X 0,Y 305.233,Z 194.017,A -85,B 0,C 180,E1 -16140.431,E2 -16140.431} C_VEL
LIN {X 0,Y 305.433,Z 190.506,A -85,B 0,C 180,E1 -16144.068,E2 -16144.068} C_VEL
LIN {X 0,Y 305.394,Z 189.541,A -85,B 0,C 180,E1 -16145.118,E2 -16145.118} C_VEL
LIN {X 0,Y 305.428,Z 189.439,A -85,B 0,C 180,E1 -16148.523,E2 -16148.523} C_VEL
LIN {X 0,Y 305.451,Z 189.435,A -85,B 0,C 180,E1 -16152.584,E2 -16152.584} C_VEL
LIN {X 0,Y 305.477,Z 189.432,A -85,B 0,C 180,E1 -16156.353,E2 -16156.353} C_VEL
LIN {X 0,Y 305.468,Z 189.432,A -85,B 0,C 180,E1 -16159.893,E2 -16159.893} C_VEL
LIN {X 0,Y 305.466,Z 189.433,A -85,B 0,C 180,E1 -16163.628,E2 -16163.628} C_VEL
LIN {X 0,Y 305.446,Z 189.437,A -85,B 0,C 180,E1 -16166.48,E2 -16166.48} C_VEL
LIN {X 0,Y 305.475,Z 189.434,A -85,B 0,C 180,E1 -16170.948,E2 -16170.948} C_VEL
LIN {X 0,Y 305.55,Z 189.423,A -85,B 0,C 180,E1 -16174.085,E2 -16174.085} C_VEL
LIN {X 0,Y 305.519,Z 189.416,A -85,B 0,C 180,E1 -16178.404,E2 -16178.404} C_VEL
LIN {X 0,Y 305.554,Z 189.414,A -85,B 0,C 180,E1 -16181.439,E2 -16181.439} C_VEL
LIN {X 0,Y 305.624,Z 189.413,A -85,B 0,C 180,E1 -16185.347,E2 -16185.347} C_VEL
LIN {X 0,Y 305.554,Z 189.42,A -85,B 0,C 180,E1 -16187.176,E2 -16187.176} C_VEL
LIN {X 0,Y 304.902,Z 189.503,A -85,B 0,C 180,E1 -16188.278,E2 -16188.278} C_VEL
LIN {X 0,Y 302.117,Z 189.85,A -85,B 0,C 180,E1 -16190.076,E2 -16190.076} C_VEL
LIN {X 0,Y 299.784,Z 190.14,A -85,B 0,C 180,E1 -16191.533,E2 -16191.533} C_VEL
LIN {X 0,Y 298.823,Z 190.26,A -85,B 0,C 180,E1 -16192.661,E2 -16192.661} C_VEL
LIN {X 0,Y 298.766,Z 190.266,A -85,B 0,C 180,E1 -16193.042,E2 -16193.042} C_VEL
LIN {X 0,Y 298.809,Z 190.259,A -85,B 0,C 180,E1 -16197.303,E2 -16197.303} C_VEL
LIN {X 0,Y 298.953,Z 190.247,A -85,B 0,C 180,E1 -16200,E2 -16200} C_VEL
LIN {X 0,Y 298.829,Z 190.259,A -85,B 0,C 180,E1 -16202.696,E2 -16202.696} C_VEL
LIN {X 0,Y 298.772,Z 190.266,A -85,B 0,C 180,E1 -16206.754,E2 -16206.754} C_VEL
LIN {X 0,Y 298.655,Z 190.285,A -85,B 0,C 180,E1 -16209.481,E2 -16209.481} C_VEL
LIN {X 0,Y 298.523,Z 190.3,A -85,B 0,C 180,E1 -16213.616,E2 -16213.616} C_VEL
LIN {X 0,Y 298.502,Z 190.301,A -85,B 0,C 180,E1 -16216.411,E2 -16216.411} C_VEL
LIN {X 0,Y 298.51,Z 190.301,A -85,B 0,C 180,E1 -16219.668,E2 -16219.668} C_VEL
LIN {X 0,Y 298.451,Z 190.307,A -85,B 0,C 180,E1 -16223.598,E2 -16223.598} C_VEL
LIN {X 0,Y 298.468,Z 190.307,A -85,B 0,C 180,E1 -16226.576,E2 -16226.576} C_VEL
LIN {X 0,Y 298.399,Z 190.309,A -85,B 0,C 180,E1 -16229.643,E2 -16229.643} C_VEL
LIN {X 0,Y 298.375,Z 190.32,A -85,B 0,C 180,E1 -16232.803,E2 -16232.803} C_VEL
LIN {X 0,Y 298.446,Z 190.311,A -85,B 0,C 180,E1 -16236.815,E2 -16236.815} C_VEL
LIN {X 0,Y 298.438,Z 190.31,A -85,B 0,C 180,E1 -16241.253,E2 -16241.253} C_VEL
LIN {X 0,Y 298.519,Z 190.406,A -85,B 0,C 180,E1 -16244.696,E2 -16244.696} C_VEL
LIN {X 0,Y 299.272,Z 195.101,A -85,B 0,C 180,E1 -16248.892,E2 -16248.892} C_VEL
LIN {X 0,Y 299.831,Z 199.355,A -85,B 0,C 180,E1 -16252.456,E2 -16252.456} C_VEL
LIN {X 0,Y 299.811,Z 202.772,A -85,B 0,C 180,E1 -16255.13,E2 -16255.13} C_VEL
LIN {X 0,Y 299.127,Z 207.81,A -85,B 0,C 180,E1 -16258.88,E2 -16258.88} C_VEL
LIN {X 0,Y 298.369,Z 213.044,A -85,B 0,C 180,E1 -16262.66,E2 -16262.66} C_VEL
LIN {X 0,Y 297.82,Z 217.718,A -85,B 0,C 180,E1 -16265.985,E2 -16265.985} C_VEL
LIN {X 0,Y 300.817,Z 230.971,A -85,B 0,C 180,E1 -16266.806,E2 -16266.806} C_VEL
LIN {X 0,Y 302.893,Z 243.357,A -85,B 0,C 180,E1 -16267.786,E2 -16267.786} C_VEL
LIN {X 0,Y 304.133,Z 255.173,A -85,B 0,C 180,E1 -16268.925,E2 -16268.925} C_VEL
LIN {X 0,Y 304.527,Z 262.515,A -85,B 0,C 180,E1 -16269.749,E2 -16269.749} C_VEL
LIN {X 0,Y 302.876,Z 274.304,A -85,B 0,C 180,E1 -16271.221,E2 -16271.221} C_VEL
LIN {X 0,Y 301.337,Z 284.815,A -85,B 0,C 180,E1 -16272.886,E2 -16272.886} C_VEL
LIN {X 0,Y 299.968,Z 293.989,A -85,B 0,C 180,E1 -16274.72,E2 -16274.72} C_VEL
LIN {X 0,Y 298.719,Z 302.132,A -85,B 0,C 180,E1 -16276.741,E2 -16276.741} C_VEL
LIN {X 0,Y 297.88,Z 307.667,A -85,B 0,C 180,E1 -16278.433,E2 -16278.433} C_VEL
LIN {X 0,Y 297.215,Z 313.085,A -85,B 0,C 180,E1 -16280.474,E2 -16280.474} C_VEL
LIN {X 0,Y 296.796,Z 317.315,A -85,B 0,C 180,E1 -16282.518,E2 -16282.518} C_VEL
LIN {X 0,Y 296.551,Z 320.478,A -85,B 0,C 180,E1 -16284.562,E2 -16284.562} C_VEL
LIN {X 0,Y 296.529,Z 322.055,A -85,B 0,C 180,E1 -16285.924,E2 -16285.924} C_VEL
LIN {X 0,Y 296.533,Z 323.205,A -85,B 0,C 180,E1 -16287.284,E2 -16287.284} C_VEL
LIN {X 0,Y 296.518,Z 324.252,A -85,B 0,C 180,E1 -16290.001,E2 -16290.001} C_VEL
LIN {X 0,Y 296.485,Z 324.195,A -85,B 0,C 180,E1 -16291.359,E2 -16291.359} C_VEL
LIN {X 0,Y 296.526,Z 323.739,A -85,B 0,C 180,E1 -16292.718,E2 -16292.718} C_VEL
LIN {X 0,Y 296.532,Z 321.565,A -85,B 0,C 180,E1 -16295.44,E2 -16295.44} C_VEL
LIN {X 0,Y 296.794,Z 318.852,A -85,B 0,C 180,E1 -16297.484,E2 -16297.484} C_VEL
LIN {X 0,Y 297.273,Z 315.125,A -85,B 0,C 180,E1 -16299.526,E2 -16299.526} C_VEL
LIN {X 0,Y 297.995,Z 310.286,A -85,B 0,C 180,E1 -16301.564,E2 -16301.564} C_VEL
LIN {X 0,Y 299.07,Z 304.192,A -85,B 0,C 180,E1 -16303.591,E2 -16303.591} C_VEL
LIN {X 0,Y 300.515,Z 296.625,A -85,B 0,C 180,E1 -16305.601,E2 -16305.601} C_VEL
LIN {X 0,Y 301.826,Z 288.682,A -85,B 0,C 180,E1 -16307.315,E2 -16307.315} C_VEL
LIN {X 0,Y 303.594,Z 278.411,A -85,B 0,C 180,E1 -16309.085,E2 -16309.085} C_VEL
LIN {X 0,Y 305.392,Z 267.748,A -85,B 0,C 180,E1 -16310.545,E2 -16310.545} C_VEL
LIN {X 0,Y 305.925,Z 262.15,A -85,B 0,C 180,E1 -16311.212,E2 -16311.212} C_VEL
LIN {X 0,Y 305.068,Z 251.839,A -85,B 0,C 180,E1 -16312.377,E2 -16312.377} C_VEL
LIN {X 0,Y 303.368,Z 240.182,A -85,B 0,C 180,E1 -16313.494,E2 -16313.494} C_VEL
LIN {X 0,Y 300.747,Z 227.601,A -85,B 0,C 180,E1 -16314.495,E2 -16314.495} C_VEL
LIN {X 0,Y 298.156,Z 217.524,A -85,B 0,C 180,E1 -16315.198,E2 -16315.198} C_VEL
LIN {X 0,Y 298.997,Z 211.454,A -85,B 0,C 180,E1 -16319.577,E2 -16319.577} C_VEL
LIN {X 0,Y 299.756,Z 206.298,A -85,B 0,C 180,E1 -16323.432,E2 -16323.432} C_VEL
LIN {X 0,Y 300.097,Z 203.225,A -85,B 0,C 180,E1 -16325.835,E2 -16325.835} C_VEL
LIN {X 0,Y 299.993,Z 200.118,A -85,B 0,C 180,E1 -16328.374,E2 -16328.374} C_VEL
LIN {X 0,Y 299.564,Z 196.654,A -85,B 0,C 180,E1 -16331.345,E2 -16331.345} C_VEL
LIN {X 0,Y 298.828,Z 192.564,A -85,B 0,C 180,E1 -16335.126,E2 -16335.126} C_VEL
LIN {X 0,Y 298.421,Z 190.315,A -85,B 0,C 180,E1 -16337.384,E2 -16337.384} C_VEL
LIN {X 0,Y 298.393,Z 190.317,A -85,B 0,C 180,E1 -16341.005,E2 -16341.005} C_VEL
LIN {X 0,Y 298.406,Z 190.316,A -85,B 0,C 180,E1 -16343.929,E2 -16343.929} C_VEL
LIN {X 0,Y 298.38,Z 190.322,A -85,B 0,C 180,E1 -16347.198,E2 -16347.198} C_VEL
LIN {X 0,Y 298.407,Z 190.315,A -85,B 0,C 180,E1 -16350.618,E2 -16350.618} C_VEL
LIN {X 0,Y 298.462,Z 190.307,A -85,B 0,C 180,E1 -16353.476,E2 -16353.476} C_VEL
